// TIA Portal V16 program export: 5 tag tables, 70 data types, 8 data blocks, 77 code blocks (in call order from the OBs), 35 instance data blocks

VAR_GLOBAL   // PLC tag table "Default tag table"
   Tag_1 AT %M66.0 : Bool;
   Tag_2 AT %M60.0 : Bool;
   Tag_3 AT %M60.1 : Bool;
   Tag_4 AT %M60.2 : Bool;
   Tag_5 AT %M60.3 : Bool;
   Tag_6 AT %M70.0 : Bool;
   Tag_7 AT %M1.0 : Bool;
   Tag_8 AT %M1.1 : Bool;
   Tag_9 AT %M1.2 : Bool;
   Tag_10 AT %M70.1 : Bool;
   Tag_11 AT %M60.5 : Bool;
   Tag_12 AT %IW0 : Word;
   Tag_13 AT %IW2 : Word;
   Tag_14 AT %IW4 : Word;
   Tag_15 AT %M66.3 : Bool;
   Tag_16 AT %M17.0 : Bool;
   Tag_17 AT %M1717.0 : Bool;
   adım1 AT %M0.0 : Bool;
   step1 AT %M0.1 : Bool;
   step2 AT %M0.2 : Bool;
   step3 AT %M0.3 : Bool;
   step4 AT %M0.4 : Bool;
   step5 AT %M0.5 : Bool;
   Tag_18 AT %M170.0 : Bool;
   Tag_19 AT %M170.1 : Bool;
   step6 AT %M0.6 : Bool;
   step7 AT %M0.7 : Bool;
   Tag_20 AT %M1717.2 : Bool;
   Tag_21 AT %MD100 : DWord;
END_VAR

VAR_GLOBAL   // PLC tag table "LSimaHydTO_Constants"
END_VAR
VAR_GLOBAL CONSTANT   // user constants
   LSIMAHYD_PROFILE_POINTS_UPPER_LIMIT : Int := 20;   // Upper limit of the points in the force profile
   LSIMAHYD_VCHAR_POINTS_UPPER_LIMIT : Int := 40;   // Upper limit of the points in the valve characteristic
END_VAR

VAR_GLOBAL   // PLC tag table "SimaHydTO_HydAxisAnalog2_Interface"
   HydAxisAnalog_2_Sensor1_Interface_AddressIn AT %I1400.0 : "PD_TEL83_IN";   //    {ExternalWritable false}
   HydAxisAnalog_2_ForceSensor AT %IW1052 : Int;   //    {ExternalWritable false}
   HydAxisAnalog_2_Sensor1_Interface_AddressOut AT %Q1400.0 : "PD_TEL83_OUT";   //    {ExternalWritable false}
   HydAxisAnalog_2_OutputValue AT %QW2 : Int;   //    {ExternalWritable false}
END_VAR

VAR_GLOBAL   // PLC tag table "SimaHydTO_HydAxisAnalog_Interface"
   HydAxisAnalog_Sensor1_Interface_AddressIn AT %I1200.0 : "PD_TEL83_IN";   //    {ExternalWritable false}
   HydAxisAnalog_ForceSensor AT %IW1050 : Int;   //    {ExternalWritable false}
   HydAxisAnalog_Sensor1_Interface_AddressOut AT %Q1200.0 : "PD_TEL83_OUT";   //    {ExternalWritable false}
   HydAxisAnalog_OutputValue AT %QW0 : Int;   //    {ExternalWritable false}
END_VAR

VAR_GLOBAL   // PLC tag table "SimaHydTO_HydAxisServo_Interface"
   HydAxisServo_Actor_Interface_AddressIn AT %I1100.0 : "PD_TEL2_IN";   //    {ExternalWritable false}
   HydAxisServo_Sensor1_Interface_AddressIn AT %I1150.0 : "PD_TEL81_IN";   //    {ExternalWritable false}
   HydAxisServo_ForceSensor AT %IW1020 : Int;   //    {ExternalWritable false}
   HydAxisServo_Actor_Interface_AddressOut AT %Q1100.0 : "PD_TEL2_OUT";   //    {ExternalWritable false}
   HydAxisServo_Sensor1_Interface_AddressOut AT %Q1150.0 : "PD_TEL81_OUT";   //    {ExternalWritable false}
END_VAR

TYPE "LSimaHydTO_typeActor"
TITLE = LSimaHydTO_typeActor
// Actor configuration
// stored: IsFailsafeCompliant false
   STRUCT
      InverseDirection { S7_SetPoint := 'True'} : Bool := FALSE;   // Inversion of the setpoint if TRUE
      BiDirectional { S7_SetPoint := 'True'} : Bool := TRUE;   // Positive and negative outputs
      SubstituteValue { S7_SetPoint := 'True'} : LReal := 0.0;   // Substitute Output Value if disabled
      MaxDerivative { S7_SetPoint := 'True'} : LReal := 10000.0;   // Limit of changes at the manipulated variable
      DirectionValves { S7_SetPoint := 'True'} : "LSimaHydTO_typeActorDirectionValves";
   END_STRUCT;
END_TYPE

TYPE "LSimaHydTO_typeActorDirectionValves"
TITLE = LSimaHydTO_typeActorDirectionValves
// Settings of the direction valves control
// stored: IsFailsafeCompliant false
   STRUCT
      WaitTimeByDirectionChange { S7_SetPoint := 'True'} : LReal := 0.0;   // Waiting time between switching the digital valve valveForward and valveBackward for a direction change [s]
      DelayTimeValveForward { S7_SetPoint := 'True'} : LReal := 0.0;   // Reaction time for digital valve [s]
      DelayTimeValveBackward { S7_SetPoint := 'True'} : LReal := 0.0;   // Reaction time for digital valve [s]
      ValvesOffMode { S7_SetPoint := 'True'} : DInt := 0;   // 0: keep digital valves on after ramp down / 1: switch off digital valves after ramp down
      DisplacementForce { S7_SetPoint := 'True'} : Bool := FALSE;   // 1: force control by displacement ( inverse direction), e.g. die cushion
   END_STRUCT;
END_TYPE

TYPE "LSimaHydTO_typeAxisData"
TITLE = LSimaHydTO_typeAxisData
// Axis data
// stored: IsFailsafeCompliant false
   STRUCT
      Velocity : LReal := 0.0;   // Velocity setpoint
      Acceleration : LReal := 0.0;   // Setpoint acceleration
      Position : LReal := 0.0;   // Position setpoint
      Force : LReal := 0.0;   // Force setpoint
      ActualVelocity : LReal := 0.0;   // Actual velocity
      ActualSpeed : LReal := 0.0;   // Actual speed of the motor (only with PROFIdrive drive type)
      ActualAcceleration : LReal := 0.0;   // Actual acceleration
      ActualPosition : LReal := 0.0;   // Actual position
      ActualForce : LReal := 0.0;   // Actual force
      Actor { S7_SetPoint := 'True'} : "LSimaHydTO_typeActor";   // Actor configuration
      ValveCharacteristic { S7_SetPoint := 'True'} : "LSimaHydTO_typeValveCharacteristic";   // Valve characteristic
      ForceLimits { S7_SetPoint := 'True'} : "LSimaHydTO_typeForceLimits";   // Force limits
      Pressure_A_Transducer { S7_SetPoint := 'True'} : "LSimaHydTO_typeTransducer";   // Piston side pressure transducer configuration
      Pressure_B_Transducer { S7_SetPoint := 'True'} : "LSimaHydTO_typeTransducer";   // Piston rod side pressure transducer configuration
      PositionControl { S7_SetPoint := 'True'} : "LSimaHydTO_typePositionControl";   // Position control configuration data
      ForceControl { S7_SetPoint := 'True'} : "LSimaHydTO_typeForceControl";   // Force control configuration data
      DynamicAxisModel { S7_SetPoint := 'True'} : "LSimaHydTO_typeDynamicAxisModel";   // Settings of the balancing filter
      SmoothingFilter { S7_SetPoint := 'True'} : "LSimaHydTO_typeSmoothingFilter";   // Settings of the smoothing filter
      StatusActor { S7_SetPoint := 'True'} : "LSimaHydTO_typeStatusActor";   // Indicates the status of actor data
      StatusVChar { S7_SetPoint := 'True'} : "LSimaHydTO_typeStatusVChar";   // Indicates the status of valve characteristic data
      Status_A_Transducer { S7_SetPoint := 'True'} : "LSimaHydTO_typeStatusTransducer";   // Indicates the status of piston side pressure transducer data
      Status_B_Transducer { S7_SetPoint := 'True'} : "LSimaHydTO_typeStatusTransducer";   // Indicates the status of piston rod side pressure transducer data
      StatusServo { S7_SetPoint := 'True'} : "LSimaHydTO_typeStatusServo";   // Indicates the status of position control
      StatusForce { S7_SetPoint := 'True'} : "LSimaHydTO_typeStatusForce";   // Indicates the status of force control
      StatusForceProfile { S7_SetPoint := 'True'} : "LSimaHydTO_typeStatusForceProfile";   // Indicates the status of a force profile processing
      ErrorWord : DWord;   // Error information
      ErrorDetail { S7_SetPoint := 'True'} : "LSimaHydTO_typeErrorDetail";   // Error Details
      "Name" { S7_SetPoint := 'True'} : WString[24];   // Name displayed on HMI
      TO_Axis : DB_ANY;   // Number of connected technology object (TO)
      DataInitialized : Bool;   // Axis data completely initialized
      Internal { S7_SetPoint := 'True'} : "LSimaHydTO_typeInternal";   // Internal axis data
   END_STRUCT;
END_TYPE

TYPE "LSimaHydTO_typeDynamicAxisModel"
TITLE = LSimaHydTO_typeDynamicAxisModel
// Settings of the balancing filter
// stored: IsFailsafeCompliant false
   STRUCT
      VelocityTimeConstant { S7_SetPoint := 'True'} : LReal;   // Speed control loop substitute time [s]
      ForceTimeConstant { S7_SetPoint := 'True'} : LReal;   // Force control loop substitute time [s]
   END_STRUCT;
END_TYPE

TYPE "LSimaHydTO_typeDynamicLimits"
TITLE = LSimaHydTO_typeDynamicLimits
// Dynamic limits
// stored: IsFailsafeCompliant false
   STRUCT
      MaxVelocity { S7_SetPoint := 'True'} : LReal := 500.0;   // Maximum permissible velocity of the axis
      MaxAcceleration { S7_SetPoint := 'True'} : LReal := 10000.0;   // Maximum permissible acceleration of the axis
      MaxDeceleration { S7_SetPoint := 'True'} : LReal := 10000.0;   // Maximum permissible deceleration of the axis
      MaxJerk { S7_SetPoint := 'True'} : LReal := 200000.0;   // Maximum permissible jerk on the axis/ not used yet
   END_STRUCT;
END_TYPE

TYPE "LSimaHydTO_typeErrorDetail"
TITLE = LSimaHydTO_typeErrorDetail
// Error Details
// stored: IsFailsafeCompliant false
   STRUCT
      Number : UDInt;   // Alarm number
      Reaction : DInt;   // Effective alarm reaction
   END_STRUCT;
END_TYPE

TYPE "LSimaHydTO_typeForceControl"
TITLE = LSimaHydTO_typeForceControl
// Force control configuration data
// stored: IsFailsafeCompliant false
   STRUCT
      SmoothingTimeByChangeDifference { S7_SetPoint := 'True'} : LReal;   // Time constant for smoothing manipulated variable jumps
      PreControl { S7_SetPoint := 'True'} : LReal := 0.0;   // Weighting factor of the precontrol Kpc [%]
      Stiffness { S7_SetPoint := 'True'} : LReal;   // Stiffness of the system, should be > 0.0 if preControl is used
      ProportionalGain { S7_SetPoint := 'True'} : LReal := 1.0;   // Proportional gain Kp
      IntegralTime { S7_SetPoint := 'True'} : LReal;   // Active integral action time Ti [s]
      DerivativeTime { S7_SetPoint := 'True'} : LReal;   // Active derivative action time Td [s]
      DecayTime { S7_SetPoint := 'True'} : LReal := 0.0;   // Decay time constant of the DT1 component [s]
      OutputUppLimit { S7_SetPoint := 'True'} : LReal := 10000.0;   // Manipulated value high limit
      OutputLowLimit { S7_SetPoint := 'True'} : LReal := -10000.0;   // Manipulated value low limit
      SmoothSwitching { S7_SetPoint := 'True'} : Bool := TRUE;   // Switching mode to force control, if TRUE, initial command value of the force controller will be presetted for edgeless valve setpoint
      InvertSetpoint { S7_SetPoint := 'True'} : Bool;   // Invert output of controller if TRUE
   END_STRUCT;
END_TYPE

TYPE "LSimaHydTO_typeForceLimits"
TITLE = LSimaHydTO_typeForceLimits
// Force limits
// stored: IsFailsafeCompliant false
   STRUCT
      MaxForce { S7_SetPoint := 'True'} : LReal := 100.0;   // Maximum force
      MaxForceRamp { S7_SetPoint := 'True'} : LReal := 10000.0;   // Force increase limitation
   END_STRUCT;
END_TYPE

TYPE "LSimaHydTO_typeInternal"
TITLE = LSimaHydTO_typeInternal
// Internal axis data
// stored: IsFailsafeCompliant false
   STRUCT
      Control { S7_SetPoint := 'True'} : "LSimaHydTO_typeInternalControl";   // Command structure, use for axis control
      MotionData { S7_SetPoint := 'True'} : "LSimaHydTO_typeInternalMotionData";   // Motion command data
      PositionLimits_SW { S7_SetPoint := 'True'} : "LSimaHydTO_typePositionLimits";   // Software position limit switch
      UnitsCorrection { S7_SetPoint := 'True'} : "LSimaHydTO_typeInternalUnitsCorrection";   // Correction of units
      CommandIDPool { ExternalAccessible := 'False'; ExternalVisible := 'False'; ExternalWritable := 'False'} : UDInt;   // Source for unique command ID's
   END_STRUCT;
END_TYPE

TYPE "LSimaHydTO_typeInternalCmdTracking"
TITLE = LSimaHydTO_typeInternalCmdTracking
// Command tracking
// stored: IsFailsafeCompliant false
   STRUCT
      CommandID : UDInt := 0;   // Command ID for tracking
      State : Word := 0;   // Command state
   END_STRUCT;
END_TYPE

TYPE "LSimaHydTO_typeInternalControl"
TITLE = LSimaHydTO_typeInternalControl
// Command structure, use for axis control
// stored: IsFailsafeCompliant false
   STRUCT
      AckError : Bool;   // Acknowledge error of axis
      ExecuteForceLimiting : Bool;   // Rising edge starts force limiting defined by ForceCommand
      ExecuteForceControl : Bool;   // Rising edge starts force control defined by ForceCommand
      RequestForward : Bool;   // request to open direction valve forward
      RequestBackward : Bool;   // request to open direction valve backward
      ForceCommand { S7_SetPoint := 'True'} : "LSimaHydTO_typeInternalControlForceCmd";   // Defines force command
      DirectOutput { S7_SetPoint := 'True'} : "LSimaHydTO_typeInternalControlDirectOutput";
   END_STRUCT;
END_TYPE

TYPE "LSimaHydTO_typeInternalControlDirectOutput"
TITLE = LSimaHydTO_typeInternalControlDirectOutput
// Manual output control
// stored: IsFailsafeCompliant false
   STRUCT
      activate : Bool;   // enables direct setting of output
      jogForward : Bool;   // direct output is active in positive direction if TRUE
      jogBackward : Bool;   // direct output is active in negative direction if TRUE
      commandValueForward : LReal := 5.0;   // direct output value in positive direction [%]
      commandValueBackward : LReal := 5.0;   // direct output value in negative direction [%]
      commandValueRamp : LReal := 100.0;   // Ramp for command value [%/s]
      offset : LReal := 0.0;   // Manipulated variable as drift compensation [%]
      safetyDistance : LReal := 50.0;   // Safety distance to avoid passing over the min. and max. positions [mm]
      commandID : UDInt;   // commanID for tracking
   END_STRUCT;
END_TYPE

TYPE "LSimaHydTO_typeInternalControlForceCmd"
TITLE = LSimaHydTO_typeInternalControlForceCmd
// Defines force command
// stored: IsFailsafeCompliant false
   STRUCT
      mode : DInt;   // 0: deactivate / 1: activate immediately / 2: starting from the time a condition is met.
      forceProfileMode : DInt;   // 0: with force value / 1: profile is a function of time / 2: profile is a function of position
      conditionMode : DInt := 1;   // 1: based on time / 2: based on position / 3: based on force/pressure
      compareMode : DInt := 1;   // 1: Value greater than or equal to ConditionValue / 2: Value less than ConditionValue
      conditionValue : LReal;   // comparison value for switching condition
      clampingMonitoring : Bool;   // TRUE: end stop detection is activated, motion stops after detection
      followingErrorDeviation : LReal;   // Required following error for recognition of the endstop
      forceValue : LReal;   // Force setpoint
      forceRamp : LReal;   // Force setpoint increase
      velocityLimitingValue : LReal;   // Rate limiting value during pressure control, the dynamic response of the pressure Value > 0.0 Use the specified value
      commandID : UDInt;   // commanID for tracking
   END_STRUCT;
END_TYPE

TYPE "LSimaHydTO_typeInternalMotionData"
TITLE = LSimaHydTO_typeInternalMotionData
// Motion command data
// stored: IsFailsafeCompliant false
   STRUCT
      PositionControlled : Bool := FALSE;   // Activates position controller
      ForceLimited : Bool := FALSE;   // Enable force limiting
      ForceControlled : Bool := FALSE;   // Enable force control
      RampingForward : Bool;   // enable signal for ramping in positive direction
      RampingBackward : Bool;   // enable signal for ramping in negative direction
      ForceCmdTracking { S7_SetPoint := 'True'} : "LSimaHydTO_typeInternalCmdTracking";   // Force command tracking
      DirectOutput { S7_SetPoint := 'True'} : "LSimaHydTO_typeInternalStatusDirectOutput";
   END_STRUCT;
END_TYPE

TYPE "LSimaHydTO_typeInternalStatusDirectOutput"
TITLE = LSimaHydTO_typeInternalStatusDirectOutput
// Manual output control
// stored: IsFailsafeCompliant false
   STRUCT
      active : Bool;   // displays activity of manual output operation
      rampingDown : Bool;   // ramping down due to positioning limits
      minSafetyPositionOverrun : Bool;   // the min. safety position was passed
      maxSafetyPositionOverrun : Bool;   // the max. safety position was passed
      QOutputValue : LReal;
      cmdTracking { S7_SetPoint := 'True'} : "LSimaHydTO_typeInternalCmdTracking";
   END_STRUCT;
END_TYPE

TYPE "LSimaHydTO_typeInternalUnitsCorrection"
TITLE = LSimaHydTO_typeInternalUnitsCorrection
// stored: IsFailsafeCompliant false
   STRUCT
      velFactor : LReal := 1.0;
      accFactor : LReal := 1.0;
   END_STRUCT;
END_TYPE

TYPE "LSimaHydTO_typeMeasuredValues"
TITLE = LSimaHydTO_typeMeasuredValues
// Measurement results
// stored: IsFailsafeCompliant false
   STRUCT
      forward { S7_SetPoint := 'True'} : "LSimaHydTO_typeVCharMeasured";   // measured values in positive direction
      backward { S7_SetPoint := 'True'} : "LSimaHydTO_typeVCharMeasured";   // measured values in negative direction
   END_STRUCT;
END_TYPE

TYPE "LSimaHydTO_typeMeasurementConfig"
TITLE = LSimaHydTO_typeMeasurementConfig
// Configuration of the measurement function
// stored: IsFailsafeCompliant false
   STRUCT
      waitTimeMeasurement { S7_SetPoint := 'True'} : DInt := 100;   // Waiting time after ramping [ms]
      maxMeasurementTime { S7_SetPoint := 'True'} : DInt := 200;   // Measurement time [ms]
      offset { S7_SetPoint := 'True'} : LReal;   // Manipulated variable as drift compensation [%]
      safetyDistance { S7_SetPoint := 'True'} : LReal;   // Safety distance to avoid passing over the min. and max. positions
      forward { S7_SetPoint := 'True'} : "LSimaHydTO_typeMeasurementQOutput";   // Structure to define the manipulated variable
      backward { S7_SetPoint := 'True'} : "LSimaHydTO_typeMeasurementQOutput";   // Structure to define the manipulated variable
      numberOfRetryMeasurement { S7_SetPoint := 'True'} : Int := 1;   // Number of repeat attempts to measure the velocity, this parameter should be greater than / equal to 1
   END_STRUCT;
END_TYPE

TYPE "LSimaHydTO_typeMeasurementQOutput"
TITLE = LSimaHydTO_typeMeasurementQOutput
// Structure to define the manipulated variable
// stored: IsFailsafeCompliant false
   STRUCT
      enableMeasurement { S7_SetPoint := 'True'} : Bool := TRUE;   // Enables measurement in this direction
      maxVelocity { S7_SetPoint := 'True'} : Real := 500.0;   // Velocity limit in this direction
      setpointForMovement { S7_SetPoint := 'True'} : Real := 40.0;   // Substitute value for movements if a measurement is not active [%]
      ramp { S7_SetPoint := 'True'} : Real := 100.0;   // manipulated variable – increase/decrease [%/s]
      minQOutputValue { S7_SetPoint := 'True'} : Real;   // start measurement with this value
      fineRange { S7_SetPoint := 'True'} : "LSimaHydTO_typeMeasurementQOutputRange";   // measurement in the fine area
      coarseRange { S7_SetPoint := 'True'} : "LSimaHydTO_typeMeasurementQOutputRange";   // measurement in the coarse area
   END_STRUCT;
   // fineRange.maxQOutputValue := 40.0;
   // fineRange.numberOfPoints := 10;
   // coarseRange.maxQOutputValue := 100.0;
   // coarseRange.numberOfPoints := 10;
END_TYPE

TYPE "LSimaHydTO_typeMeasurementQOutputRange"
TITLE = LSimaHydTO_typeMeasurementQOutputRange
// stored: IsFailsafeCompliant false
   STRUCT
      maxQOutputValue { S7_SetPoint := 'True'} : Real;   // incremented up to this value
      numberOfPoints { S7_SetPoint := 'True'} : Int;   // number of points for this range
   END_STRUCT;
END_TYPE

TYPE "LSimaHydTO_typeMotionVector"
TITLE = LSimaHydTO_typeMotionVector
// Values of a motion vector
// stored: IsFailsafeCompliant false
   STRUCT
      Position : LReal;   // Position
      Velocity : LReal;   // Velocity
      Acceleration : LReal;   // Acceleration
   END_STRUCT;
END_TYPE

TYPE "LSimaHydTO_typePositionControl"
TITLE = LSimaHydTO_typePositionControl
// Position control configuration data
// stored: IsFailsafeCompliant false
   STRUCT
      SmoothingTimeByChangeDifference { S7_SetPoint := 'True'} : LReal;   // Time constant for smoothing manipulated variable jumps [s]
      PreControl { S7_SetPoint := 'True'} : LReal := 100.0;   // Weighting factor of the precontrol Kpc [%]
      ProportionalGain { S7_SetPoint := 'True'} : LReal := 10.0;   // Proportional gain Kp [1/s]
      IntegralTime { S7_SetPoint := 'True'} : LReal;   // Active integral action time Ti [s]
      DerivativeTime { S7_SetPoint := 'True'} : LReal;   // Active derivative action time Td [s]
      DecayTime { S7_SetPoint := 'True'} : LReal := 0.0;   // Decay time constant of the DT1 component [s]
      OutputUppLimit { S7_SetPoint := 'True'} : LReal := 10000.0;   // Manipulated value high limit [unit/s]
      OutputLowLimit { S7_SetPoint := 'True'} : LReal := -10000.0;   // Manipulated value low limit [unit/s]
   END_STRUCT;
END_TYPE

TYPE "LSimaHydTO_typePositionLimits"
TITLE = LSimaHydTO_typePositionLimits
// Software position limit switch
// stored: IsFailsafeCompliant false
   STRUCT
      Active { S7_SetPoint := 'True'} : Bool := TRUE;   // FALSE: Monitoring disabled / TRUE: Monitoring enabled
      MinPosition { S7_SetPoint := 'True'} : LReal := -1000000000000.0;   // Position of negative SW limit switch
      MaxPosition { S7_SetPoint := 'True'} : LReal := 1000000000000.0;   // Position of positive SW limit switch
   END_STRUCT;
END_TYPE

TYPE "LSimaHydTO_typeProfile"
TITLE = LSimaHydTO_typeProfile
// Configuration for the profile point
// stored: IsFailsafeCompliant false
   STRUCT
      LeadingValue { S7_SetPoint := 'True'} : Array[0.."LSIMAHYD_PROFILE_POINTS_UPPER_LIMIT"] of Real;   // Input values array
      Value { S7_SetPoint := 'True'} : Array[0.."LSIMAHYD_PROFILE_POINTS_UPPER_LIMIT"] of Real;   // Output values array
      MaxIdx { S7_SetPoint := 'True'} : Int;   // Max used index in arrays
   END_STRUCT;
END_TYPE

TYPE "LSimaHydTO_typeSmoothingFilter"
TITLE = LSimaHydTO_typeSmoothingFilter
// Settings of the smoothing filter
// stored: IsFailsafeCompliant false
   STRUCT
      VelocityFilter { S7_SetPoint := 'True'} : LReal := 0.0;   // Time constant for actual velocity smoothing filter [s]
      AccelerationFilter { S7_SetPoint := 'True'} : LReal := 0.0;   // Time constant for actual acceleration smoothing filter [s]
   END_STRUCT;
END_TYPE

TYPE "LSimaHydTO_typeStatusActor"
TITLE = LSimaHydTO_typeStatusActor
// Indicates the status of actor data
// stored: IsFailsafeCompliant false
   STRUCT
      SetPoint : LReal := 0.0;   // Manipulated variable
      AddSetPoint : LReal := 0.0;   // Additional setpoint
      QOutputValue : LReal := 0.0;   // Output value in relation to Q-output [%]
      Enabled : Bool;   // Output is enabled
      ValveForward : Bool := FALSE;   // Control bit for positive direction
      ValveBackward : Bool := FALSE;   // Control bit for negative direction
   END_STRUCT;
END_TYPE

TYPE "LSimaHydTO_typeStatusForce"
TITLE = LSimaHydTO_typeStatusForce
// Indicates the status of force control
// stored: IsFailsafeCompliant false
   STRUCT
      ForceLimitingCommand { ExternalWritable := 'False'} : Bool;   // TRUE: Axis is in force limiting mode; FALSE: Axis isn't in force limiting mode/ SimaHyd only
      InLimitation { ExternalWritable := 'False'} : Bool;   // TRUE: Axis is operating at the force limit; FALSE: axis is not operating at the force limit/ SimaHyd only
      InClamping { ExternalWritable := 'False'} : Bool;   // TRUE: Axis is clamped at a fixed stop; FALSE: Axis is not clamped at a fixed stop
      ForceControl { ExternalWritable := 'False'} : Bool;   // TRUE: Axis is in force control mode; FALSE: Axis isn't in force control mode/ SimaHyd only
      TargetForce { ExternalWritable := 'False'} : LReal;   // Target force
      ForceDerivedValue { ExternalWritable := 'False'} : LReal;   // Rate-of-change limiting for the force setpoint
      PreControlValue { ExternalWritable := 'False'} : LReal;   // Force precontrol value
      BalancedForce { ExternalWritable := 'False'} : LReal;   // Force after the balancing filter
      ControlDifference { ExternalWritable := 'False'} : LReal;   // Control error
      ControlOutput { ExternalWritable := 'False'} : LReal;   // Control variable
   END_STRUCT;
END_TYPE

TYPE "LSimaHydTO_typeStatusForceProfile"
TITLE = LSimaHydTO_typeStatusForceProfile
// Indicates the status of a force profile processing
// stored: IsFailsafeCompliant false
   STRUCT
      ActualProfile : UInt := 0;   // Currently effective force profile DB number
      ForceProfileMode : DInt := 0;   // 0: with force value / 1: profile is a function of time / 2: profile is a function of position
      Active : Bool := FALSE;   // Activation status of a command for specifying the force profile
      State : DInt := 0;   // Execution state: 0: inactive / 1: in interpolation / 2: on profile / 3: profile end
      BaseValue : LReal := 0.0;   // Current reference value
      ProfileValue : LReal := 0.0;   // Profile value for the base value
   END_STRUCT;
END_TYPE

TYPE "LSimaHydTO_typeStatusServo"
TITLE = LSimaHydTO_typeStatusServo
// Indicates the status of position control
// stored: IsFailsafeCompliant false
   STRUCT
      BalancedPosition { ExternalWritable := 'False'} : LReal;   // Position after the balancing filter
      ControlDifference { ExternalWritable := 'False'} : LReal;   // Control error
   END_STRUCT;
END_TYPE

TYPE "LSimaHydTO_typeStatusTransducer"
TITLE = LSimaHydTO_typeStatusTransducer
// Indicates the status of transducer data
// stored: IsFailsafeCompliant false
   STRUCT
      RawValue : Word;   // Raw data of analog input
      PressureValue : LReal;   // actual pressure In pressure units
      ForceValue : LReal;   // actual force In force units
      Error : Bool := FALSE;   // Indicates error of transducer
   END_STRUCT;
END_TYPE

TYPE "LSimaHydTO_typeStatusVChar"
TITLE = LSimaHydTO_typeStatusVChar
// Indicates the status of valve characteristic data
// stored: IsFailsafeCompliant false
   STRUCT
      ActualVChar : UInt := 0;   // Currently effective valve characteristic DB number
   END_STRUCT;
END_TYPE

TYPE "LSimaHydTO_typeTransducer"
TITLE = LSimaHydTO_typeTransducer
// Pressure transducer configuration
// stored: IsFailsafeCompliant false
   STRUCT
      HWReference { S7_SetPoint := 'True'} : Int := 16#6C00;   // Normalization of the raw value for 100%. Distinction between a SIMATIC or a SINAMICS periphery: SIMATIC = 27648, SINAMICS = 16384
      NominalPressure { S7_SetPoint := 'True'} : LReal := 400.0;   // Nominal pressure of transducer, e.g. 400 [bar]
      Area { S7_SetPoint := 'True'} : LReal := 1.0;   // Area [mm2] or [in2]
      Offset { S7_SetPoint := 'True'} : LReal := 0.0;   // Offset in pressure units
      FilterTime { S7_SetPoint := 'True'} : LReal := 0.0;   // Smoothing filter
      ErrorValue { S7_SetPoint := 'True'} : Word := 16#7FFF;   // Error signal
   END_STRUCT;
END_TYPE

TYPE "LSimaHydTO_typeVCharData"
TITLE = LSimaHydTO_typeVCharData
// Valve characteristic description
// stored: IsFailsafeCompliant false
   STRUCT
      QOutput { S7_SetPoint := 'True'} : Array[0.."LSIMAHYD_VCHAR_POINTS_UPPER_LIMIT"] of Real;   // Output values array
      Velocity { S7_SetPoint := 'True'} : Array[0.."LSIMAHYD_VCHAR_POINTS_UPPER_LIMIT"] of Real;   // Velocity values array
      VelocityLimitPositive { S7_SetPoint := 'True'} : Real;   // Max velocity in positive direction
      VelocityLimitNegative { S7_SetPoint := 'True'} : Real;   // Max velocity in negative direction
      ZeroZonePositive { S7_SetPoint := 'True'} : Real;   // Overlapping zone of valve in positive direction
      ZeroZoneNegative { S7_SetPoint := 'True'} : Real;   // Overlapping zone of valve in negative direction
      MaxIdx { S7_SetPoint := 'True'} : Int;   // Max used index in arrays
      "Name" { S7_SetPoint := 'True'} : WString[24];   // Symbolic name displayed on HMI for index of array
   END_STRUCT;
END_TYPE

TYPE "LSimaHydTO_typeVCharMeasured"
TITLE = LSimaHydTO_typeVCharMeasured
// Measured Values in one direction
// stored: IsFailsafeCompliant false
   STRUCT
      qOutput : Array[0.."LSIMAHYD_VCHAR_POINTS_UPPER_LIMIT"] of Real;   // manipulated variable
      velocity : Array[0.."LSIMAHYD_VCHAR_POINTS_UPPER_LIMIT"] of Real;   // velocity
      maxVelocity : Real;   // max. measured velocity
      minQOutput : Real;   // min. manipulated variable
      maxQOutput : Real;   // max. manipulated variable
      maxIndexMeasurement : Int;   // measurement was made up to this index
      coarseBegin : Real;   // coarse area begins by this index
   END_STRUCT;
END_TYPE

TYPE "LSimaHydTO_typeValveCharacteristic"
TITLE = LSimaHydTO_typeValveCharacteristic
// Valve characteristic
// stored: IsFailsafeCompliant false
   STRUCT
      DB_NUMBER { S7_SetPoint := 'True'} : UInt;   // Number of DB of type LSimaHydTO_typeVCharData with valve profile data
      SmoothChangeTime { S7_SetPoint := 'True'} : Real;   // Filter time for smooth changing
      SmoothingMode { S7_SetPoint := 'True'} : Int;   // Filter mode for smooth changing: 0: T1 / 1: ramping with constant ramp / 2: ramping with time
   END_STRUCT;
END_TYPE

TYPE "SimaHydTO_typeAxesArray"
TITLE = SimaHydTO_typeAxesArray
// Axis array of HMI axis selection
// stored: IsFailsafeCompliant false
   STRUCT
      axisData { ExternalAccessible := 'False'; ExternalVisible := 'False'; ExternalWritable := 'False'} : DB_ANY;   // DB number of hydraulic axis DB (HydAxisTO)
      basicControl { ExternalAccessible := 'False'; ExternalVisible := 'False'; ExternalWritable := 'False'; S7_SetPoint := 'True'} : "SimaHydTO_typeHMIConnectionBasicAxisControlCommand";   // HMI -> PLC: Axis commands of technology object via PLCopen functions
      directOutputControl { ExternalAccessible := 'False'; ExternalVisible := 'False'; ExternalWritable := 'False'; S7_SetPoint := 'True'} : "SimaHydTO_typeIHMIConnectionBasicAxisControlDirectOutput";
      VCharMeasurement { ExternalAccessible := 'False'; ExternalVisible := 'False'; ExternalWritable := 'False'; S7_SetPoint := 'True'} : "SimaHydTO_typeAxesArrayVCharMeasurement";
      advancedControl { ExternalAccessible := 'False'; ExternalVisible := 'False'; ExternalWritable := 'False'; S7_SetPoint := 'True'} : "SimaHydTO_typeHMIConnectionAdvancedAxisControlCommand";   // Advanced axis commands of technology object via PLCopen functions
      initialized { ExternalAccessible := 'False'; ExternalVisible := 'False'; ExternalWritable := 'False'} : Bool;   // Axis data initialized
   END_STRUCT;
END_TYPE

TYPE "SimaHydTO_typeAxesArrayVCharMeasurement"
TITLE = SimaHydTO_typeAxesArrayVCharMeasurement
// Axis array of HMI axis selection
// stored: IsFailsafeCompliant false
   STRUCT
      requestForward { ExternalAccessible := 'False'; ExternalVisible := 'False'; ExternalWritable := 'False'} : Bool;   // Switches the digital valves to move in the positive direction
      requestBackward { ExternalAccessible := 'False'; ExternalVisible := 'False'; ExternalWritable := 'False'} : Bool;   // Switches the digital valves to move in the negative direction
      enableRampingForward { ExternalAccessible := 'False'; ExternalVisible := 'False'; ExternalWritable := 'False'} : Bool := True;   // Enable ramping of Q-Output value (voltage) in positivedirection
      enableRampingBackward { ExternalAccessible := 'False'; ExternalVisible := 'False'; ExternalWritable := 'False'} : Bool := True;   // Enable ramping of Q-Output value (voltage) in negative direction
   END_STRUCT;
END_TYPE

TYPE "SimaHydTO_typeHMIConnection"
TITLE = SimaHydTO_typeHMIConnection
// HMI connection interface data block
// stored: IsFailsafeCompliant false
   STRUCT
      AxisData { S7_SetPoint := 'True'} : "SimaHydTO_typeHMIConnectionAxisData";
      AxisToData { S7_SetPoint := 'True'} : "SimaHydTO_typeHMIConnectionAxisToData";
      AxisSelector { S7_SetPoint := 'True'} : "SimaHydTO_typeHMIConnectionAxisSelector";
      BasicAxisControl { S7_SetPoint := 'True'} : "SimaHydTO_typeHMIConnectionBasicAxisControl";
      GetCharacteristics { S7_SetPoint := 'True'} : "SimaHydTO_typeHMIConnectionGetCharacteristicInterface";
      HmiData { S7_SetPoint := 'True'} : "SimaHydTO_typeHMIConnectionHmiData";
      VCharEditor { S7_SetPoint := 'True'} : "SimaHydTO_typeHMIConnectionVCharEditor";
      AdvancedAxisControl { S7_SetPoint := 'True'} : "SimaHydTO_typeHMIConnectionAdvancedAxisControl";
      ParameterSettings { S7_SetPoint := 'True'} : "SimaHydTO_typeHMIConnectionParameterSettings";
   END_STRUCT;
END_TYPE

TYPE "SimaHydTO_typeHMIConnectionAdvancedAxisControl"
TITLE = SimaHydTO_typeHMIConnectionAdvancedAxisControl
// HMI interface: Advanced axis control
// stored: IsFailsafeCompliant false
   STRUCT
      Command { S7_SetPoint := 'True'} : "SimaHydTO_typeHMIConnectionAdvancedAxisControlCommand";   // Command (HMI -> PLC)
      Status { S7_SetPoint := 'True'} : "SimaHydTO_typeHMIConnectionAdvancedAxisControlStatus";   // Status (PLC -> HMI)
   END_STRUCT;
END_TYPE

TYPE "SimaHydTO_typeHMIConnectionAdvancedAxisControlCommand"
TITLE = SimaHydTO_typeHMIConnectionAdvancedAxisControlCommand
// HMI interface: Advanced axis control
// stored: IsFailsafeCompliant false
   STRUCT
      moveRelativeExecute : Bool;   // MC_MoveRelative: Start job with a positive edge
      moveRelativeDistance : LReal;   // Distance of relative movement
      moveAbsoluteExecute : Bool;   // MC_MoveAbsolute: Start job with a positive edge
      moveAbsolutePosition : LReal;   // Target position of absolute movement
      moveAbsoluteDirection : Int := 3;   // Direction of absolute movement: 0: Positive direction / 1: Negative direction / 3: Shortest direction
      haltExecute : Bool;   // MC_Halt: Start job with a positive edge
      haltAbortAcceleration : Bool;   // Acceleration control: False: The current acceleration at the start of the job is reduced using the configured jerk. Afterwards, the deceleration builds up / True: The acceleration is set to 0.0 at the start of the job, and the deceleration immediately builds up.
      Velocity : LReal := -1.0;   // Velocity of movement
      Acceleration : LReal := -1.0;   // Acceleration of movement
      Deceleration : LReal := -1.0;   // Deceleration of movement
      Jerk : LReal := -1.0;   // Jerk of movement
   END_STRUCT;
END_TYPE

TYPE "SimaHydTO_typeHMIConnectionAdvancedAxisControlStatus"
TITLE = SimaHydTO_typeHMIConnectionAdvancedAxisControlStatus
// HMI interface: Advanced axis control
// stored: IsFailsafeCompliant false
   STRUCT
      moveRelativeDone : Bool;   // MC_MoveRelative: Job is completed
      moveRelativeBusy : Bool;   // MC_MoveRelative: Job is running
      moveAbsoluteDone : Bool;   // MC_MoveAbsolute: Job is completed
      moveAbsoluteBusy : Bool;   // MC_MoveAbsolute: Job is running
      haltDone : Bool;   // MC_Halt: Job is running
      haltBusy : Bool;   // MC_Halt: Job is running
      commandAborted : Bool;   // The job was aborted by another job during execution (see also StatusID)
      error : Bool;   // An error occurred during execution of the job. The job is rejected. The cause of the error can be found in the "ErrorID" parameter.
      errorID : Word;   // ErrorID of motion control instruction (see also StatusID)
      statusID : Int;   // Additional specification of affected Motion control instruction of CommandAborted or Error: 0: No instruction / 1: MC_MoveRelative / 2: MC_MoveAbsolute / 3: MC_Halt
   END_STRUCT;
END_TYPE

TYPE "SimaHydTO_typeHMIConnectionAxisData"
TITLE = SimaHydTO_typeHMIConnectionAxisData
// Axis data
// stored: IsFailsafeCompliant false
   STRUCT
      Velocity : LReal := 0.0;   // Velocity setpoint
      Acceleration : LReal := 0.0;   // Setpoint acceleration
      Position : LReal := 0.0;   // Position setpoint
      Force : LReal := 0.0;   // Force setpoint
      ActualVelocity : LReal := 0.0;   // Actual velocity
      ActualSpeed : LReal := 0.0;   // Actual speed of the motor (only with PROFIdrive drive type)
      ActualAcceleration : LReal := 0.0;   // Actual acceleration
      ActualPosition : LReal := 0.0;   // Actual position
      ActualForce : LReal := 0.0;   // Actual force
      StatusActor { S7_SetPoint := 'True'} : "LSimaHydTO_typeStatusActor";   // Indicates the status of actor data
      StatusVChar { S7_SetPoint := 'True'} : "LSimaHydTO_typeStatusVChar";   // Indicates the status of valve characteristic data
      Status_A_Transducer { S7_SetPoint := 'True'} : "LSimaHydTO_typeStatusTransducer";   // Indicates the status of piston side pressure transducer data
      Status_B_Transducer { S7_SetPoint := 'True'} : "LSimaHydTO_typeStatusTransducer";   // Indicates the status of piston rod side pressure transducer data
      StatusServo { S7_SetPoint := 'True'} : "LSimaHydTO_typeStatusServo";   // Indicates the status of position control
      StatusForce { S7_SetPoint := 'True'} : "LSimaHydTO_typeStatusForce";   // Indicates the status of force control
      StatusForceProfile { S7_SetPoint := 'True'} : "LSimaHydTO_typeStatusForceProfile";   // Indicates the status of a force profile processing
      ErrorWord : DWord;   // Error information
      ErrorDetail { S7_SetPoint := 'True'} : "LSimaHydTO_typeErrorDetail";   // Error Details
      "Name" : WString[24];   // Name displayed on HMI
   END_STRUCT;
END_TYPE

TYPE "SimaHydTO_typeHMIConnectionAxisSelector"
TITLE = SimaHydTO_typeHMIConnectionAxisSelector
// HMI interface: Axis selection of axis array
// stored: IsFailsafeCompliant false
   STRUCT
      Command { S7_SetPoint := 'True'} : "SimaHydTO_typeHMIConnectionAxisSelectorCommand";   // Data: HMI -> PLC
      Status { S7_SetPoint := 'True'} : "SimaHydTO_typeHMIConnectionAxisSelectorStatus";   // Data: PLC -> HMI
   END_STRUCT;
END_TYPE

TYPE "SimaHydTO_typeHMIConnectionAxisSelectorCommand"
TITLE = SimaHydTO_typeHMIConnectionAxisSelectorCommand
// HMI interface: Axis selection of axis array - Command (HMI -> PLC)
// stored: IsFailsafeCompliant false
   STRUCT
      previousObject : Bool;
      nextObject : Bool;
      executeDirectIndexSelection : Bool;
      directIndexSelection : Int;
   END_STRUCT;
END_TYPE

TYPE "SimaHydTO_typeHMIConnectionAxisSelectorStatus"
TITLE = SimaHydTO_typeHMIConnectionAxisSelectorStatus
// HMI interface: Axis selection of axis array - Status (PLC -> HMI)
// stored: IsFailsafeCompliant false
   STRUCT
      actualAxisIndex : Int;   // Actual selected array index
      selectedAxis : DB_ANY;   // DB number of actual selected hydraulic axis
      selectedTO_Axis : DB_ANY;   // DB/TO number of actual selected technology object axis
      selectedVChar : DB_ANY;   // DB number of actual selected valve characteristics
      selectedAxisInteger : UInt;   // DB number of actual selected hydraulic axis as integer value
      selectedAxisTOInteger : UInt;   // DB/TO number of actual selected technology object as integer value
      selectedVCharInteger : UInt;   // DB number of actual selected valve characteristics as integer value
      selectedAxisName : WString[24];   // Name of actual selected hydraulic axis
      selectedVCharName : WString[24];   // Name of active VChat of selected hydraulic axis
      selectedTypeOfAxis : Int;   // 0: No axis / 1: Speed axis / 2: Positioning axis / 3: Synchronous axis / 4: External encoder
      selectionChanged : Bool;   // axis selection is changed
      dataValid : Bool;   // Selected data valid
      dataError : Bool;   // Error of data selection
   END_STRUCT;
END_TYPE

TYPE "SimaHydTO_typeHMIConnectionAxisToData"
TITLE = SimaHydTO_typeHMIConnectionAxisToData
// HMI interface: Technology object axis diagnostic words
// stored: IsFailsafeCompliant false
   STRUCT
      statusWord : DWord;
      warningWord : DWord;
      errorWord : DWord;
      errorDetail { S7_SetPoint := 'True'} : "SimaHydTO_typeHMIConnectionAxisToDataErrorDetail";
      axisUnits { S7_SetPoint := 'True'} : "SimaHydTO_typeHMIConnectionAxisToDataAxisUnits";
      typeOfAxis : Int;   // 0: No axis / 1: Speed axis / 2: Positioning axis / 3: Synchronous axis / 4: External encoder
   END_STRUCT;
END_TYPE

TYPE "SimaHydTO_typeHMIConnectionAxisToDataAxisUnits"
TITLE = SimaHydTO_typeHMIConnectionAxisToDataAxisUnits
// HMI interface: Technology object axis units
// stored: IsFailsafeCompliant false
   STRUCT
      lengthUnit : UDInt := 0;
      velocityUnit : UDInt := 0;
      forceUnit : UDInt := 0;
      timeUnit : UDInt := 1054;
   END_STRUCT;
END_TYPE

TYPE "SimaHydTO_typeHMIConnectionAxisToDataErrorDetail"
TITLE = SimaHydTO_typeHMIConnectionAxisToDataErrorDetail
// HMI interface: Technology object axis error detail
// stored: IsFailsafeCompliant false
   STRUCT
      number : UDInt;   // Error number
      reaction : DInt;   // Error reaction
   END_STRUCT;
END_TYPE

TYPE "SimaHydTO_typeHMIConnectionBasicAxisControl"
TITLE = SimaHydTO_typeHMIConnectionBasicAxisControl
// HMI interface: Basic axis control (LAxisBasics)
// stored: IsFailsafeCompliant false
   STRUCT
      Command { S7_SetPoint := 'True'} : "SimaHydTO_typeHMIConnectionBasicAxisControlCommand";
      Status { S7_SetPoint := 'True'} : "SimaHydTO_typeHMIConnectionBasicAxisControlStatus";
      ControlDirectOutput { S7_SetPoint := 'True'} : "SimaHydTO_typeIHMIConnectionBasicAxisControlDirectOutput";
      StatusDirectOutput { S7_SetPoint := 'True'} : "SimaHydTO_typeHMIConnectionBasicAxislStatusDirectOutput";
   END_STRUCT;
END_TYPE

TYPE "SimaHydTO_typeHMIConnectionBasicAxisControlCommand"
TITLE = SimaHydTO_typeHMIConnectionBasicAxisControlCommand
// HMI interface: Basic axis control (LAxisBasics) - Command (HMI -> PLC)
// stored: IsFailsafeCompliant false
   STRUCT
      powerEnable : Bool;   // MC_Power: 0: The technology object is disabled / 1: The technology object is enabled
      powerStartMode : DInt := 1;   // 0: Enable axis not position-controlled / 1: Enable axis position-controlled
      powerStopMode : Int := 0;   // 0: Emergency stop / 1: Immediate stop / 2: Stop with maximum dynamic values
      resetExecute : Bool;   // MC_Reset: Start job with a positive edge
      resetFBExecute : Bool;   // LSimaHyd_MC_Reset: Start job with a positive edge
      resetRestart : Bool := false;   // 0: Acknowledgment of queued technology alarms / 1: Reinitialization of the technology object and acknowledgment of pending technology alarms
      homeExecute : Bool;   // MC_Home: Start job with a positive edge
      homePosition : LReal;   // The specified value is used according to the selected "Mode".
      homeMode : Int;   // 0: Direct homing (absolute) / 1: Direct homing (relative) / 2: Passive homing / 3: Active homing / 4: Reserved / 5: Active homing (<TO>.Homing.HomePosition) / 6: Absolute encoder adjustment (relative) / 7: Absolute encoder adjustment (absolute) / 8: Passive homing / 9: Abort passive homing / 10: Passive homing (<TO>.Homing.HomePosition)
      jogForward : Bool;   // MC_MoveJog: As long as the parameter is TRUE, the axis moves in the positive direction
      jogBackward : Bool;   // MC_MoveJog: As long as the parameter is TRUE, the axis moves in the negative direction
      jogVelocity : LReal := 100.0;   // Velocity setpoint / speed setpoint for the motion
      jogAcceleration : LReal := -1.0;   // Acceleration of jog movement
      jogDeceleration : LReal := -1.0;   // Deceleration of jog movement
      jogJerk : LReal := -1.0;   // Jerk of jog movement
      jogPositionControlled : Bool := true;   // 0: Non position-controlled operation / 1: Position-controlled mode - The parameter applies as long as the MC_MoveJog command is executed. After this, the setting of MC_Power applies again.
   END_STRUCT;
END_TYPE

TYPE "SimaHydTO_typeHMIConnectionBasicAxisControlStatus"
TITLE = SimaHydTO_typeHMIConnectionBasicAxisControlStatus
// HMI interface: Basic axis control (LAxisBasics) - Status (PLC -> HMI)
// stored: IsFailsafeCompliant false
   STRUCT
      powerStatus : Bool;   // MC_Power: 0: Technology object disabled / 1: Technology object enabled
      powerBusy : Bool;   // MC_Power: Job is running
      resetDone : Bool;   // MC_Reset: Error has been acknowledged or Restart has been executed.
      resetBusy : Bool;   // MC_Reset: Job is running
      resetFBDone : Bool;   // LSimaHyd_MC_Reset: Error has been acknowledged or Restart has been executed.
      resetFBBusy : Bool;   // LSimaHyd_MC_Reset: Job is running
      homeDone : Bool;   // MC_Home: Job is completed
      homeBusy : Bool;   // MC_Home: Job is running
      jogInVelocity : Bool;   // MC_MoveJog: The velocity setpoint / speed setpoint was reached and will be maintained
      jogBusy : Bool;   // MC_MoveJog: Job is running
      commandAborted : Bool;   // The job was aborted by another job during execution (see also StatusID)
      error : Bool;   // An error occurred during execution of the job. The job is rejected. The cause of the error can be found in the "ErrorID" parameter.
      errorID : Word;   // ErrorID of motion control instruction (see also StatusID)
      statusID : Int;   // Additional specification of affected Motion control instruction of CommandAborted or Error: 0: No instruction / 1: MC_Power / 2: MC_Reset / 3: MC_Home / 4: MC_MoveJog
   END_STRUCT;
END_TYPE

TYPE "SimaHydTO_typeHMIConnectionBasicAxislStatusDirectOutput"
TITLE = SimaHydTO_typeHMIConnectionBasicAxislStatusDirectOutput
// Direct output status
// stored: IsFailsafeCompliant false
   STRUCT
      active : Bool;   // displays activity of direct output operation
      rampingDown : Bool;   // ramping down due to positioning limits
      minSafetyPositionOverrun : Bool;   // the min. safety position was passed
      maxSafetyPositionOverrun : Bool;   // the max. safety position was passed
   END_STRUCT;
END_TYPE

TYPE "SimaHydTO_typeHMIConnectionGetCharacteristicInterface"
TITLE = SimaHydTO_typeHMIConnectionGetCharacteristicInterface
// Function block interface of FB "GetCharacteristics"
// stored: IsFailsafeCompliant false
   STRUCT
      Command { S7_SetPoint := 'True'} : "SimaHydTO_typeHMIConnectionGetCharacteristicInterfaceCommand";   // HMI -> PLC: Commands to function block GetCharacteristics
      Status { S7_SetPoint := 'True'} : "SimaHydTO_typeHMIConnectionGetCharacteristicInterfaceStatus";   // PLC -> HMI: Status of function block GetCharacteristics
      ConfigData { S7_SetPoint := 'True'} : "LSimaHydTO_typeMeasurementConfig";
      MeasuredValues { S7_SetPoint := 'True'} : "LSimaHydTO_typeMeasuredValues";
   END_STRUCT;
END_TYPE

TYPE "SimaHydTO_typeHMIConnectionGetCharacteristicInterfaceCommand"
TITLE = SimaHydTO_typeHMIConnectionGetCharacteristicInterfaceCommand
// Function block command interface of FB "GetCharacteristics"
// stored: IsFailsafeCompliant false
   STRUCT
      execute : Bool;   // Start measurement
      abort : Bool;   // Stop measurement
      enableRampingForward : Bool := True;   // Enable ramping of Q-Output value (voltage) in positivedirection
      enableRampingBackward : Bool := True;   // Enable ramping of Q-Output value (voltage) in negative direction
      saveConfig : Bool;   // Save measurement configuration
      loadConfig : Bool;   // Load measurement configuration
   END_STRUCT;
END_TYPE

TYPE "SimaHydTO_typeHMIConnectionGetCharacteristicInterfaceStatus"
TITLE = SimaHydTO_typeHMIConnectionGetCharacteristicInterfaceStatus
// Function block status interface of FB "GetCharacteristics"
// stored: IsFailsafeCompliant false
   STRUCT
      qOutputValueStepForward { ExternalWritable := 'False'} : LReal;   // Last successfully measured manipulated variable in the positive direction
      qOutputValueStepBackward { ExternalWritable := 'False'} : LReal;   // Last successfully measured velocity in the negative direction
      velocityStepForward { ExternalWritable := 'False'} : LReal;   // Last successfully measured velocity in the positive direction
      velocityStepBackward { ExternalWritable := 'False'} : LReal;   // Last successfully measured velocity in the negative direction
      requestForward { ExternalWritable := 'False'} : Bool;   // Request switching to move in the positive direction
      requestBackward { ExternalWritable := 'False'} : Bool;   // Request switching to move in the negative direction
      statusMeasurement { ExternalWritable := 'False'} : Word;   // Status of current measurement
      done { ExternalWritable := 'False'} : Bool;   // The measurement was successfully completed
      busy { ExternalWritable := 'False'} : Bool;   // Measurement active
      commandAborted { ExternalWritable := 'False'} : Bool;   // Measurement function was interrupted
      error { ExternalWritable := 'False'} : Bool;   // There is an error in the FB
      status { ExternalWritable := 'False'} : Word;   // Error information or status of the block
   END_STRUCT;
END_TYPE

TYPE "SimaHydTO_typeHMIConnectionHmiData"
TITLE = SimaHydTO_typeHMIConnectionHmiData
// HMI interface: Data to display on HMI
// stored: IsFailsafeCompliant false
   STRUCT
      stateSubNavigation : Int;
      ActualPositionPercent : Int;   // Actual axis position in percent between MinPosition and MaxPosition
      SafetyDistanceAnimation : LReal;   // SafetyDistance in percent between MinPosition and MaxPosition
      MinPosition : LReal;   // Minimal position of axis (SW limit switch)
      MaxPosition : LReal;   // Maximal position of axis (SW limit switch)
      selectedAxis : Int;   // DB number of actual selected hydraulic axis
      selectedAxisTO : Int;   // DB/TO number of actual selected technology object
      selectedVChar : Int;   // DB number of actual selected valve characteristics
      VChar { S7_SetPoint := 'True'} : "SimaHydTO_typeHMIConnectionHmiDataVChar";   // Data storage of HMI VChar display
   END_STRUCT;
END_TYPE

TYPE "SimaHydTO_typeHMIConnectionHmiDataVChar"
TITLE = SimaHydTO_typeHMIConnectionHmiDataVChar
// HMI interface: Calculated positions of VHar to display on HMI
// stored: IsFailsafeCompliant false
   STRUCT
      HMI_VChar : Array[1..200] of Real;
      HMI_VChar_MinQOutput : Real;
      HMI_VChar_MaxQOutput : Real;
      HMI_VChar_MinVelocity : Real;
      HMI_VCHar_MaxVelocity : Real;
      HMI_VChar_TrendRequest : Word;
      HMI_VChar_TrendTransfer : Word;
   END_STRUCT;
END_TYPE

TYPE "SimaHydTO_typeHMIConnectionParameterSettings"
TITLE = SimaHydTO_typeHMIConnectionParameterSettings
// HMI interface: Parameter settings
// stored: IsFailsafeCompliant false
   STRUCT
      AxisData { S7_SetPoint := 'True'} : "SimaHydTO_typeHMIConnectionParameterSettingsAxisData";
      Commands { S7_SetPoint := 'True'} : "SimaHydTO_typeHMIConnectionParameterSettingsCommands";   // Data: HMI -> PLC
      Status { S7_SetPoint := 'True'} : "SimaHydTO_typeHMIConnectionParameterSettingsStatus";   // Data: PLC -> HMI
   END_STRUCT;
END_TYPE

TYPE "SimaHydTO_typeHMIConnectionParameterSettingsAxisData"
TITLE = SimaHydTO_typeHMIConnectionParameterSettingsAxisData
// Axis data
// stored: IsFailsafeCompliant false
   STRUCT
      Actor { S7_SetPoint := 'True'} : "LSimaHydTO_typeActor";   // Actor configuration
      ValveCharacteristic { S7_SetPoint := 'True'} : "LSimaHydTO_typeValveCharacteristic";   // Valve characteristic
      ForceLimits { S7_SetPoint := 'True'} : "LSimaHydTO_typeForceLimits";   // Force limits
      Pressure_A_Transducer { S7_SetPoint := 'True'} : "LSimaHydTO_typeTransducer";   // Piston side pressure transducer configuration
      Pressure_B_Transducer { S7_SetPoint := 'True'} : "LSimaHydTO_typeTransducer";   // Piston rod side pressure transducer configuration
      PositionControl { S7_SetPoint := 'True'} : "LSimaHydTO_typePositionControl";   // Position control configuration data
      ForceControl { S7_SetPoint := 'True'} : "LSimaHydTO_typeForceControl";   // Force control configuration data
      DynamicAxisModel { S7_SetPoint := 'True'} : "LSimaHydTO_typeDynamicAxisModel";   // Settings of the balancing filter
      SmoothingFilter { S7_SetPoint := 'True'} : "LSimaHydTO_typeSmoothingFilter";   // Settings of the smoothing filter
      StatusActor { S7_SetPoint := 'True'} : "LSimaHydTO_typeStatusActor";   // Indicates the status of actor data
      StatusVChar { S7_SetPoint := 'True'} : "LSimaHydTO_typeStatusVChar";   // Indicates the status of valve characteristic data
      Status_A_Transducer { S7_SetPoint := 'True'} : "LSimaHydTO_typeStatusTransducer";   // Indicates the status of piston side pressure transducer data
      Status_B_Transducer { S7_SetPoint := 'True'} : "LSimaHydTO_typeStatusTransducer";   // Indicates the status of piston rod side pressure transducer data
      StatusServo { S7_SetPoint := 'True'} : "LSimaHydTO_typeStatusServo";   // Indicates the status of position control
      StatusForce { S7_SetPoint := 'True'} : "LSimaHydTO_typeStatusForce";   // Indicates the status of force control
      StatusForceProfile { S7_SetPoint := 'True'} : "LSimaHydTO_typeStatusForceProfile";   // Indicates the status of a force profile processing
      "Name" : WString[24];   // Name displayed on HMI
      VCharName : WString[24];   // Charachteristic name displayed on HMI
   END_STRUCT;
END_TYPE

TYPE "SimaHydTO_typeHMIConnectionParameterSettingsCommands"
TITLE = SimaHydTO_typeHMIConnectionParameterSettingsCommands
// HMI interface: Parameter settings - Command (HMI -> PLC)
// stored: IsFailsafeCompliant false
   STRUCT
      Edit : Bool;
      Activate : Bool;
      Save : Bool;
      Restore : Bool;
      Abort : Bool;
      ApplyVChar : Bool;
      VCharSelector { S7_SetPoint := 'True'} : "SimaHydTO_typeHMIConnectionVCharSelectorCommand";
   END_STRUCT;
END_TYPE

TYPE "SimaHydTO_typeHMIConnectionParameterSettingsStatus"
TITLE = SimaHydTO_typeHMIConnectionParameterSettingsStatus
// HMI interface: Parameter settings - Status (PLC -> HMI)
// stored: IsFailsafeCompliant false
   STRUCT
      EditorActive : Bool;
      StateActivation : Int;   // 0: none / 1: activated / 2: error
      StateSaving : Int;   // 0: none / 1: saved / 2: error
      StateLoading : Int;   // 0: none / 1: restoreded / 2: error
      VCharSelector { S7_SetPoint := 'True'} : "SimaHydTO_typeHMIConnectionVCharSelectorStatus";
   END_STRUCT;
END_TYPE

TYPE "SimaHydTO_typeHMIConnectionVCharEditor"
TITLE = SimaHydTO_typeHMIConnectionVCharEditor
// HMI interface: VChar editor
// stored: IsFailsafeCompliant false
   STRUCT
      Command { S7_SetPoint := 'True'} : "SimaHydTO_typeHMIConnectionVCharEditorCommand";   // Data: HMI -> PLC
      Status { S7_SetPoint := 'True'} : "SimaHydTO_typeHMIConnectionVCharEditorStatus";   // Data: PLC -> HMI
      Parameter { S7_SetPoint := 'True'} : "SimaHydTO_typeHMIConnectionVCharEditorParameter";   // Data: PLC <-> HMI (Load and save)
      Table { S7_SetPoint := 'True'} : "SimaHydTO_typeHMIConnectionVCharEditorTable";   // Data table of VChar
      VCharNameToSave : WString[24];   // Name of VChar to be saved
   END_STRUCT;
END_TYPE

TYPE "SimaHydTO_typeHMIConnectionVCharEditorCommand"
TITLE = SimaHydTO_typeHMIConnectionVCharEditorCommand
// HMI interface: VChar editor - Command (HMI -> PLC)
// stored: IsFailsafeCompliant false
   STRUCT
      LoadMeasuredValues : Bool;
      LoadVChar : Bool;
      VCharLoad { S7_SetPoint := 'True'} : "SimaHydTO_typeHMIConnectionVCharSelectorCommand";
      CreateNewVChar : Bool;
      ShowPreviousRow : Bool;
      ShowNextRow : Bool;
      SaveVChar : Bool;
      SaveVCharAs : Bool;
      VCharSave { S7_SetPoint := 'True'} : "SimaHydTO_typeHMIConnectionVCharSelectorCommand";
      AbortEditor : Bool;
      DeleteRow : Bool;
      AddRow : Bool;
      SortAndDisplay : Bool;
   END_STRUCT;
END_TYPE

TYPE "SimaHydTO_typeHMIConnectionVCharEditorParameter"
TITLE = SimaHydTO_typeHMIConnectionVCharEditorParameter
// HMI interface: VChar editor
// stored: IsFailsafeCompliant false
   STRUCT
      ActualTableStartIndex : Int;
      SelectedTableIndex : Int;
      MaximumNumberOfLines : Int;
      NumberOfUsedLines : Int;
      NumberOfUsableLines : Int;
   END_STRUCT;
END_TYPE

TYPE "SimaHydTO_typeHMIConnectionVCharEditorStatus"
TITLE = SimaHydTO_typeHMIConnectionVCharEditorStatus
// HMI interface: VChar editor - Status (PLC -> HMI)
// stored: IsFailsafeCompliant false
   STRUCT
      EditorActive : Bool;
      SaveAsSelected : Bool;
      Busy : Bool;
      Error : Bool;
      VCharLoad { S7_SetPoint := 'True'} : "SimaHydTO_typeHMIConnectionVCharSelectorStatus";
      VCharSave { S7_SetPoint := 'True'} : "SimaHydTO_typeHMIConnectionVCharSelectorStatus";
   END_STRUCT;
END_TYPE

TYPE "SimaHydTO_typeHMIConnectionVCharEditorTable"
TITLE = SimaHydTO_typeHMIConnectionVCharEditorTable
// HMI interface: VChar editor
// stored: IsFailsafeCompliant false
   STRUCT
      Appearance : Array[0..20] of Int;   // 0: invisible / 1: visible / 2: selected
      Index : Array[0..20] of Int;
      Velocity : Array[0..20] of Real;
      QOutput : Array[0..20] of Real;
      VelocityLimitPositive : Real;   // Max velocity in positive direction
      VelocityLimitNegative : Real;   // Max velocity in negative direction
      ZeroZonePositive : Real;   // Overlapping zone of valve in positive direction
      ZeroZoneNegative : Real;   // Overlapping zone of valve in negative direction
   END_STRUCT;
END_TYPE

TYPE "SimaHydTO_typeHMIConnectionVCharSelectorCommand"
TITLE = SimaHydTO_typeHMIConnectionVCharSelectorCommand
// HMI interface: Hydraulic characteristics (VChar) selection of VChar array - Command (HMI -> PLC)
// stored: IsFailsafeCompliant false
   STRUCT
      previousObject : Bool;
      nextObject : Bool;
      executeDirectIndexSelection : Bool;
      directIndexSelection : Int;
   END_STRUCT;
END_TYPE

TYPE "SimaHydTO_typeHMIConnectionVCharSelectorStatus"
TITLE = SimaHydTO_typeHMIConnectionVCharSelectorStatus
// HMI interface: Hydraulic characteristics (VChar) selection of VChar array - Status (PLC -> HMI)
// stored: IsFailsafeCompliant false
   STRUCT
      actualVCharIndex : Int;   // Actual selected array index
      selectedVCharInteger : UInt;   // DB number of actual selected valve characteristics as integer value
      selectedVChar : DB_ANY;   // DB number of actual selected valve characteristics
      selectedVCharName : WString[24];   // Name of actual selected valve characteristics
      dataValid : Bool;   // Selected data valid
      dataError : Bool;   // Error of data selection
   END_STRUCT;
END_TYPE

TYPE "SimaHydTO_typeIHMIConnectionBasicAxisControlDirectOutput"
TITLE = SimaHydTO_typeIHMIConnectionBasicAxisControlDirectOutput
// Direct output control
// stored: IsFailsafeCompliant false
   STRUCT
      jogForward : Bool;   // Direct output is active in positive direction if TRUE
      jogBackward : Bool;   // Direct output is active in negative direction if TRUE
      commandValueForward : LReal := 5.0;   // Direct output value in positive direction [%]
      commandValueBackward : LReal := 5.0;   // Direct output value in negative direction [%]
      commandValueRamp : LReal := 100.0;   // Ramp for command value [%/s]
      safetyDistance : LReal := 50.0;   // Safety distance to avoid passing over the min. and max. positions
   END_STRUCT;
END_TYPE

TYPE "SimaHydTO_typeVCharArray"
TITLE = SimaHydTO_typeVCharArray
// VChar (characteristics) array of HMI VChar selection
// stored: IsFailsafeCompliant false
   STRUCT
      VChar_DB : DB_ANY;   // DB number of VChar storage
      measurementConfig { S7_SetPoint := 'True'} : "LSimaHydTO_typeMeasurementConfig";
      initialized : Bool;
   END_STRUCT;
END_TYPE

DATA_BLOCK "DENEME"   // DB3
{ S7_Optimized_Access := 'TRUE' }
VERSION : 0.1
// stored: AutoNumber true, DBAccessibleFromOPCUA true, IsOnlyStoredInLoadMemory false, IsRetainMemResEnabled false, IsWriteProtectedInAS false, MemoryReserve 100
   VAR
      VELO : Real;
      RESET : Bool;
      MoveABS : Bool;
      AbsolutePoz : Real;
      ABSvelo : Real;
      CETVEL : Real;
      HOME : Bool;
      ABSOLUTE_AUX : Real;
      OFFSET : Real;
   END_VAR
BEGIN
END_DATA_BLOCK

DATA_BLOCK "HydAxisAnalogInterface1"   // DB33150
{ S7_Optimized_Access := 'TRUE' }
FAMILY : SimaHydTO
VERSION : 1.0
// stored: AutoNumber true, DBAccessibleFromOPCUA true, IsOnlyStoredInLoadMemory false, IsRetainMemResEnabled false, IsWriteProtectedInAS false, MemoryReserve 0
   VAR
      tel81 { ExternalAccessible := 'False'; ExternalVisible := 'False'; ExternalWritable := 'False'; S7_SetPoint := 'True'} : PD_TEL81;
   END_VAR
BEGIN
END_DATA_BLOCK

DATA_BLOCK "HydAxisAnalogInterface2"   // DB33151
{ S7_Optimized_Access := 'TRUE' }
FAMILY : SimaHydTO
VERSION : 1.0
// stored: AutoNumber true, DBAccessibleFromOPCUA true, IsOnlyStoredInLoadMemory false, IsRetainMemResEnabled false, IsWriteProtectedInAS false, MemoryReserve 0
   VAR
      tel81 { ExternalAccessible := 'False'; ExternalVisible := 'False'; ExternalWritable := 'False'; S7_SetPoint := 'True'} : PD_TEL81;
   END_VAR
BEGIN
END_DATA_BLOCK

DATA_BLOCK "HydAxisDriveInterface"   // DB33152
{ S7_Optimized_Access := 'FALSE'; DB_Accessible_From_OPC_UA := 'FALSE' }
FAMILY : SimaHydTO
VERSION : 1.0
// stored: AutoNumber true, DBAccessibleFromOPCUA false, IsOnlyStoredInLoadMemory false, IsWriteProtectedInAS false
   VAR
      tel2 { ExternalAccessible := 'False'; ExternalVisible := 'False'; ExternalWritable := 'False'; S7_SetPoint := 'True'} : PD_TEL2;
      tel81 { ExternalAccessible := 'False'; ExternalVisible := 'False'; ExternalWritable := 'False'; S7_SetPoint := 'True'} : PD_TEL81;
   END_VAR
BEGIN
END_DATA_BLOCK

DATA_BLOCK "LSimaHydTO_HydAxisAnalogInterfaceTemplate"   // DB33050
TITLE = LSimaHydTO_HydAxisAnalogInterfaceTemplate
{ S7_Optimized_Access := 'TRUE'; DB_Accessible_From_OPC_UA := 'FALSE' }
AUTHOR : APC_ERLF
FAMILY : LSimaHydTO
VERSION : 1.0
// stored: AutoNumber true, DBAccessibleFromOPCUA false, IsOnlyStoredInLoadMemory false, IsRetainMemResEnabled false, IsWriteProtectedInAS false, MemoryReserve 0
   VAR
      tel81 { ExternalAccessible := 'False'; ExternalVisible := 'False'; ExternalWritable := 'False'; S7_SetPoint := 'True'} : PD_TEL81;
   END_VAR
BEGIN
END_DATA_BLOCK

DATA_BLOCK "LSimaHydTO_HydAxisDriveInterfaceTemplate"   // DB33051
TITLE = LSimaHydTO_HydAxisDriveInterfaceTemplate
{ S7_Optimized_Access := 'FALSE'; DB_Accessible_From_OPC_UA := 'FALSE' }
AUTHOR : APC_ERLF
FAMILY : LSimaHydTO
VERSION : 1.0
// stored: AutoNumber true, DBAccessibleFromOPCUA false, IsOnlyStoredInLoadMemory false, IsWriteProtectedInAS false
   VAR
      tel2 { ExternalAccessible := 'False'; ExternalVisible := 'False'; ExternalWritable := 'False'; S7_SetPoint := 'True'} : PD_TEL2;
      tel81 { ExternalAccessible := 'False'; ExternalVisible := 'False'; ExternalWritable := 'False'; S7_SetPoint := 'True'} : PD_TEL81;
   END_VAR
BEGIN
END_DATA_BLOCK

DATA_BLOCK "SimaHydTO_AxesArray"   // DB33101
TITLE = SimaHydTO_AxesArray
{ S7_Optimized_Access := 'TRUE'; DB_Accessible_From_OPC_UA := 'FALSE' }
FAMILY : SimaHydTO
VERSION : 1.0
// Array of hydraulic axes usabel in HMI
// stored: AutoNumber true, DBAccessibleFromOPCUA false, IsOnlyStoredInLoadMemory false, IsRetainMemResEnabled false, IsWriteProtectedInAS false, MemoryReserve 100
   VAR
      axes { S7_SetPoint := 'True'} : Array[0..2] of "SimaHydTO_typeAxesArray";   // Hydraulic axes of the project to be controlled via HMI
   END_VAR
BEGIN
END_DATA_BLOCK

DATA_BLOCK "SimaHydTO_VCharArray"   // DB33102
TITLE = SimaHydTO_VCharArray
{ S7_Optimized_Access := 'TRUE'; DB_Accessible_From_OPC_UA := 'FALSE' }
FAMILY : SimaHydTO
VERSION : 1.0
// Array of valve chracteristics usabel in HMI
// stored: AutoNumber true, DBAccessibleFromOPCUA false, IsOnlyStoredInLoadMemory false, IsRetainMemResEnabled false, IsWriteProtectedInAS false, MemoryReserve 100
   VAR
      VChar { S7_SetPoint := 'True'} : Array[0..12] of "SimaHydTO_typeVCharArray";   // Valve charactersitics of the project to be controlled via HMI
   END_VAR
BEGIN
   VChar[0].VChar_DB := 5001;
END_DATA_BLOCK

ORGANIZATION_BLOCK "Main"   // OB1, FBD, ProgramCycle
TITLE = "Main Program Sweep (Cycle)"
{ S7_Optimized_Access := 'TRUE' }
VERSION : 0.1
// stored: AutoNumber true, IsIECCheckEnabled false, SetENOAutomatically false
   VAR_INPUT
      Initial_Call : Bool;   // Initial call of this OB
      Remanence : Bool;   // =True, if remanent data are available
   END_VAR
BEGIN
END_ORGANIZATION_BLOCK

ORGANIZATION_BLOCK "MC-PostServo"   // OB95, LAD, PostServo
{ S7_Optimized_Access := 'TRUE' }
VERSION : 0.1
// stored: IsIECCheckEnabled false, SetENOAutomatically false
   VAR_INPUT
      Initial_Call : Bool;
      PIP_Input : Bool;
      PIP_Output : Bool;
      IO_System : USInt;
      Event_Count : Int;
      Synchronous : Bool;
      CycleTime : UDInt;
   END_VAR
   VAR_TEMP
      tempCycleTime : LReal;
      tempCycleTimeLINT : LInt;
      tempRetVal : Word;
      VELOO : Real;
      cetvel2 : Real;
   END_VAR
   VAR_TEMP   // added for the SCL form of the ladder/FBD networks
      _w1 : Bool;
      _w2 : Bool;
   END_VAR
BEGIN

REGION Network 1: Set characteristics of axis at first call
   // Initial setting of valve characteristics.
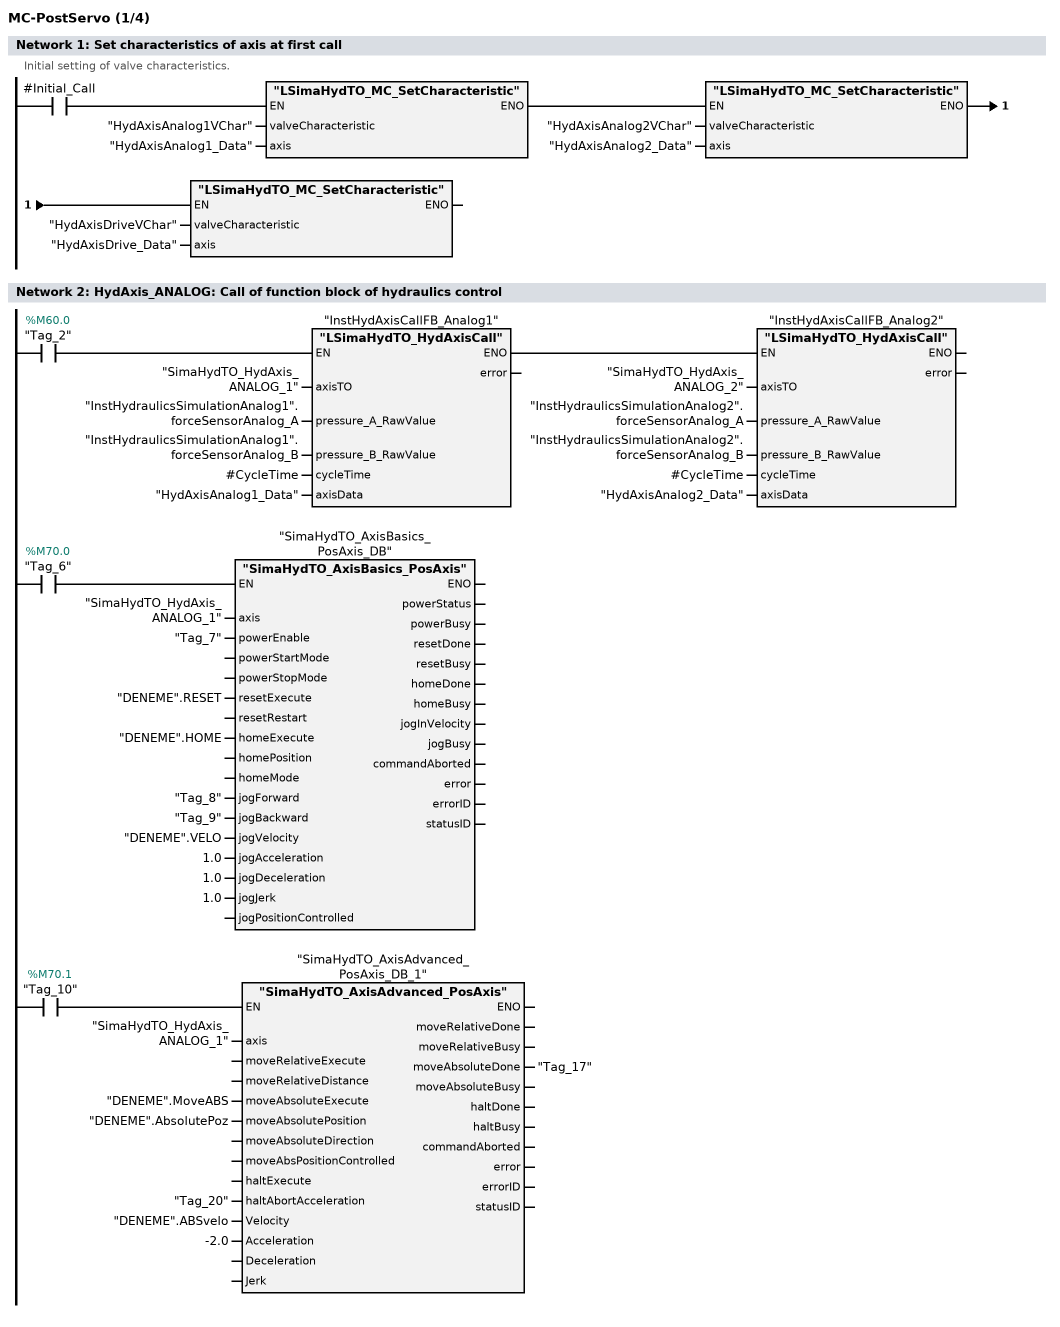
   RUNG wire#powerrail
      Contact( #Initial_Call )
      "LSimaHydTO_MC_SetCharacteristic"(valveCharacteristic := "HydAxisAnalog1VChar", axis := "HydAxisAnalog1_Data")
      "LSimaHydTO_MC_SetCharacteristic"(valveCharacteristic := "HydAxisAnalog2VChar", axis := "HydAxisAnalog2_Data")
      "LSimaHydTO_MC_SetCharacteristic"(valveCharacteristic := "HydAxisDriveVChar", axis := "HydAxisDrive_Data")
   END_RUNG
   // the same network as SCL:
   "LSimaHydTO_MC_SetCharacteristic"(EN := #Initial_Call,
                           valveCharacteristic := "HydAxisAnalog1VChar",
                           axis := "HydAxisAnalog1_Data",
                           ENO => #_w1);
   "LSimaHydTO_MC_SetCharacteristic"(EN := #_w1,
                           valveCharacteristic := "HydAxisAnalog2VChar",
                           axis := "HydAxisAnalog2_Data",
                           ENO => #_w2);
   IF #_w2 THEN
       "LSimaHydTO_MC_SetCharacteristic"(valveCharacteristic := "HydAxisDriveVChar", axis := "HydAxisDrive_Data");
   END_IF;
END_REGION

REGION Network 2: HydAxis_ANALOG: Call of function block of hydraulics control
   RUNG wire#powerrail
      Contact( "Tag_2" )
      "InstHydAxisCallFB_Analog1"(axisTO := "SimaHydTO_HydAxis_ANALOG_1", pressure_A_RawValue := "InstHydraulicsSimulationAnalog1".forceSensorAnalog_A, pressure_B_RawValue := "InstHydraulicsSimulationAnalog1".forceSensorAnalog_B, cycleTime := #CycleTime, axisData := "HydAxisAnalog1_Data", error =>)
      "InstHydAxisCallFB_Analog2"(axisTO := "SimaHydTO_HydAxis_ANALOG_2", pressure_A_RawValue := "InstHydraulicsSimulationAnalog2".forceSensorAnalog_A, pressure_B_RawValue := "InstHydraulicsSimulationAnalog2".forceSensorAnalog_B, cycleTime := #CycleTime, axisData := "HydAxisAnalog2_Data", error =>)
   END_RUNG
   RUNG wire#powerrail
      Contact( "Tag_6" )
      "SimaHydTO_AxisBasics_PosAxis_DB"(axis := "SimaHydTO_HydAxis_ANALOG_1", powerEnable := "Tag_7", powerStartMode :=, powerStopMode :=, resetExecute := "DENEME".RESET, resetRestart :=, homeExecute := "DENEME".HOME, homePosition :=, homeMode :=, jogForward := "Tag_8", jogBackward := "Tag_9", jogVelocity := "DENEME".VELO, jogAcceleration := 1.0, jogDeceleration := 1.0, jogJerk := 1.0, jogPositionControlled :=, powerStatus =>, powerBusy =>, resetDone =>, resetBusy =>, homeDone =>, homeBusy =>, jogInVelocity =>, jogBusy =>, commandAborted =>, error =>, errorID =>, statusID =>)
   END_RUNG
   RUNG wire#powerrail
      Contact( "Tag_10" )
      "SimaHydTO_AxisAdvanced_PosAxis_DB_1"(axis := "SimaHydTO_HydAxis_ANALOG_1", moveRelativeExecute :=, moveRelativeDistance :=, moveAbsoluteExecute := "DENEME".MoveABS, moveAbsolutePosition := "DENEME".AbsolutePoz, moveAbsoluteDirection :=, moveAbsPositionControlled :=, haltExecute :=, haltAbortAcceleration := "Tag_20", Velocity := "DENEME".ABSvelo, Acceleration := -2.0, Deceleration :=, Jerk :=, moveRelativeDone =>, moveRelativeBusy =>, moveAbsoluteDone => "Tag_17", moveAbsoluteBusy =>, haltDone =>, haltBusy =>, commandAborted =>, error =>, errorID =>, statusID =>)
   END_RUNG
   // the same network as SCL:
   "InstHydAxisCallFB_Analog1"(EN := "Tag_2",   // "LSimaHydTO_HydAxisCall"
                           axisTO := "SimaHydTO_HydAxis_ANALOG_1",
                           pressure_A_RawValue := "InstHydraulicsSimulationAnalog1".forceSensorAnalog_A,
                           pressure_B_RawValue := "InstHydraulicsSimulationAnalog1".forceSensorAnalog_B,
                           cycleTime := #CycleTime,
                           axisData := "HydAxisAnalog1_Data",
                           ENO => #_w1);
   IF #_w1 THEN
       "InstHydAxisCallFB_Analog2"(axisTO := "SimaHydTO_HydAxis_ANALOG_2",   // "LSimaHydTO_HydAxisCall"
                               pressure_A_RawValue := "InstHydraulicsSimulationAnalog2".forceSensorAnalog_A,
                               pressure_B_RawValue := "InstHydraulicsSimulationAnalog2".forceSensorAnalog_B,
                               cycleTime := #CycleTime,
                               axisData := "HydAxisAnalog2_Data");
   END_IF;
   IF "Tag_6" THEN
       "SimaHydTO_AxisBasics_PosAxis_DB"(axis := "SimaHydTO_HydAxis_ANALOG_1",   // "SimaHydTO_AxisBasics_PosAxis"
                               powerEnable := "Tag_7",
                               resetExecute := "DENEME".RESET,
                               homeExecute := "DENEME".HOME,
                               jogForward := "Tag_8",
                               jogBackward := "Tag_9",
                               jogVelocity := "DENEME".VELO,
                               jogAcceleration := 1.0,
                               jogDeceleration := 1.0,
                               jogJerk := 1.0);
   END_IF;
   IF "Tag_10" THEN
       "SimaHydTO_AxisAdvanced_PosAxis_DB_1"(axis := "SimaHydTO_HydAxis_ANALOG_1",   // "SimaHydTO_AxisAdvanced_PosAxis"
                               moveAbsoluteExecute := "DENEME".MoveABS,
                               moveAbsolutePosition := "DENEME".AbsolutePoz,
                               haltAbortAcceleration := "Tag_20",
                               Velocity := "DENEME".ABSvelo,
                               Acceleration := -2.0,
                               moveAbsoluteDone => "Tag_17");
   END_IF;
END_REGION

REGION Network 3: HydAxis_ANALOG: Call of function block of hydraulics axis simulation
   // The simulation uses as input signal "analogInput" the real output integer value of analog module AQ. (-27648...+27648)
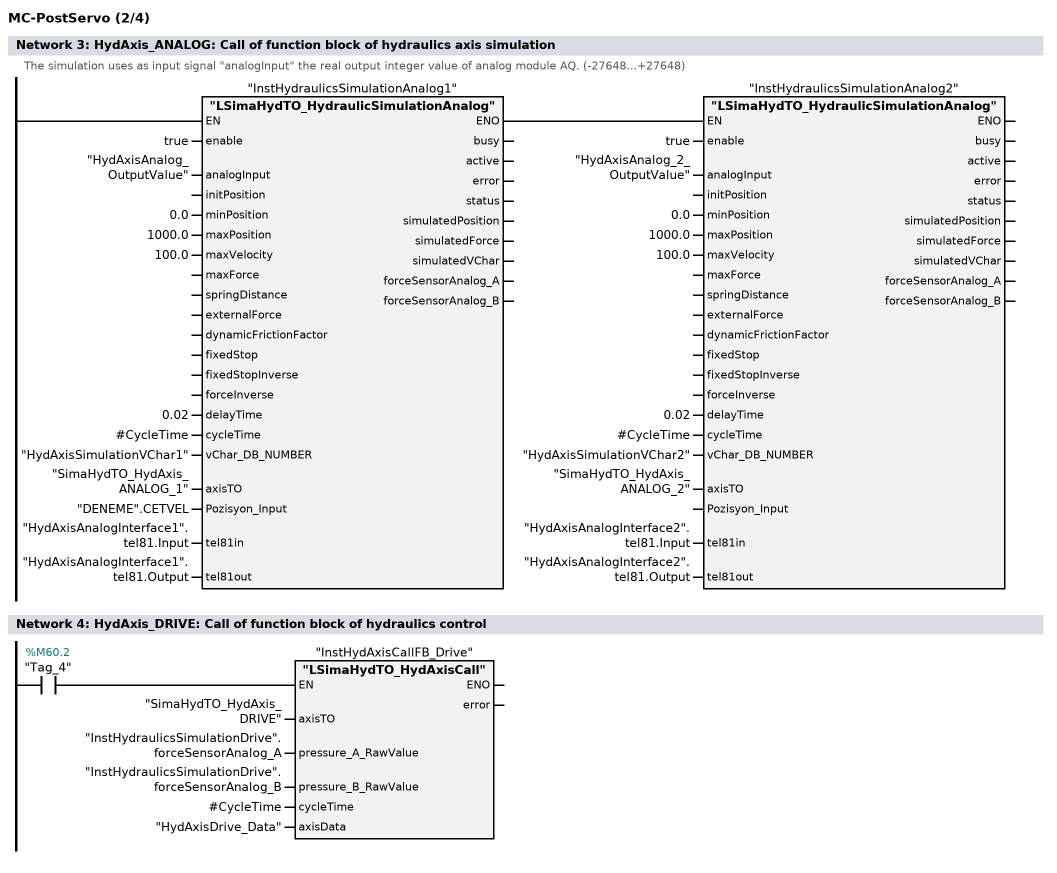
   RUNG wire#powerrail
      "InstHydraulicsSimulationAnalog1"(enable := true, analogInput := "HydAxisAnalog_OutputValue", initPosition :=, minPosition := 0.0, maxPosition := 1000.0, maxVelocity := 100.0, maxForce :=, springDistance :=, externalForce :=, dynamicFrictionFactor :=, fixedStop :=, fixedStopInverse :=, forceInverse :=, delayTime := 0.02, cycleTime := #CycleTime, vChar_DB_NUMBER := "HydAxisSimulationVChar1", axisTO := "SimaHydTO_HydAxis_ANALOG_1", Pozisyon_Input := "DENEME".CETVEL, tel81in := "HydAxisAnalogInterface1".tel81.Input, tel81out := "HydAxisAnalogInterface1".tel81.Output, busy =>, active =>, error =>, status =>, simulatedPosition =>, simulatedForce =>, simulatedVChar =>, forceSensorAnalog_A =>, forceSensorAnalog_B =>)
      "InstHydraulicsSimulationAnalog2"(enable := true, analogInput := "HydAxisAnalog_2_OutputValue", initPosition :=, minPosition := 0.0, maxPosition := 1000.0, maxVelocity := 100.0, maxForce :=, springDistance :=, externalForce :=, dynamicFrictionFactor :=, fixedStop :=, fixedStopInverse :=, forceInverse :=, delayTime := 0.02, cycleTime := #CycleTime, vChar_DB_NUMBER := "HydAxisSimulationVChar2", axisTO := "SimaHydTO_HydAxis_ANALOG_2", Pozisyon_Input :=, tel81in := "HydAxisAnalogInterface2".tel81.Input, tel81out := "HydAxisAnalogInterface2".tel81.Output, busy =>, active =>, error =>, status =>, simulatedPosition =>, simulatedForce =>, simulatedVChar =>, forceSensorAnalog_A =>, forceSensorAnalog_B =>)
   END_RUNG
   // the same network as SCL:
   "InstHydraulicsSimulationAnalog1"(enable := true,   // "LSimaHydTO_HydraulicSimulationAnalog"
                           analogInput := "HydAxisAnalog_OutputValue",
                           minPosition := 0.0,
                           maxPosition := 1000.0,
                           maxVelocity := 100.0,
                           delayTime := 0.02,
                           cycleTime := #CycleTime,
                           vChar_DB_NUMBER := "HydAxisSimulationVChar1",
                           axisTO := "SimaHydTO_HydAxis_ANALOG_1",
                           Pozisyon_Input := "DENEME".CETVEL,
                           tel81in := "HydAxisAnalogInterface1".tel81.Input,
                           tel81out := "HydAxisAnalogInterface1".tel81.Output,
                           ENO => #_w1);
   IF #_w1 THEN
       "InstHydraulicsSimulationAnalog2"(enable := true,   // "LSimaHydTO_HydraulicSimulationAnalog"
                               analogInput := "HydAxisAnalog_2_OutputValue",
                               minPosition := 0.0,
                               maxPosition := 1000.0,
                               maxVelocity := 100.0,
                               delayTime := 0.02,
                               cycleTime := #CycleTime,
                               vChar_DB_NUMBER := "HydAxisSimulationVChar2",
                               axisTO := "SimaHydTO_HydAxis_ANALOG_2",
                               tel81in := "HydAxisAnalogInterface2".tel81.Input,
                               tel81out := "HydAxisAnalogInterface2".tel81.Output);
   END_IF;
END_REGION

REGION Network 4: HydAxis_DRIVE: Call of function block of hydraulics control
   RUNG wire#powerrail
      Contact( "Tag_4" )
      "InstHydAxisCallFB_Drive"(axisTO := "SimaHydTO_HydAxis_DRIVE", pressure_A_RawValue := "InstHydraulicsSimulationDrive".forceSensorAnalog_A, pressure_B_RawValue := "InstHydraulicsSimulationDrive".forceSensorAnalog_B, cycleTime := #CycleTime, axisData := "HydAxisDrive_Data", error =>)
   END_RUNG
   // the same network as SCL:
   IF "Tag_4" THEN
       "InstHydAxisCallFB_Drive"(axisTO := "SimaHydTO_HydAxis_DRIVE",   // "LSimaHydTO_HydAxisCall"
                               pressure_A_RawValue := "InstHydraulicsSimulationDrive".forceSensorAnalog_A,
                               pressure_B_RawValue := "InstHydraulicsSimulationDrive".forceSensorAnalog_B,
                               cycleTime := #CycleTime,
                               axisData := "HydAxisDrive_Data");
   END_IF;
END_REGION

REGION Network 5: HydAxis_DRIVE: Call of function block of hydraulics axis simulation
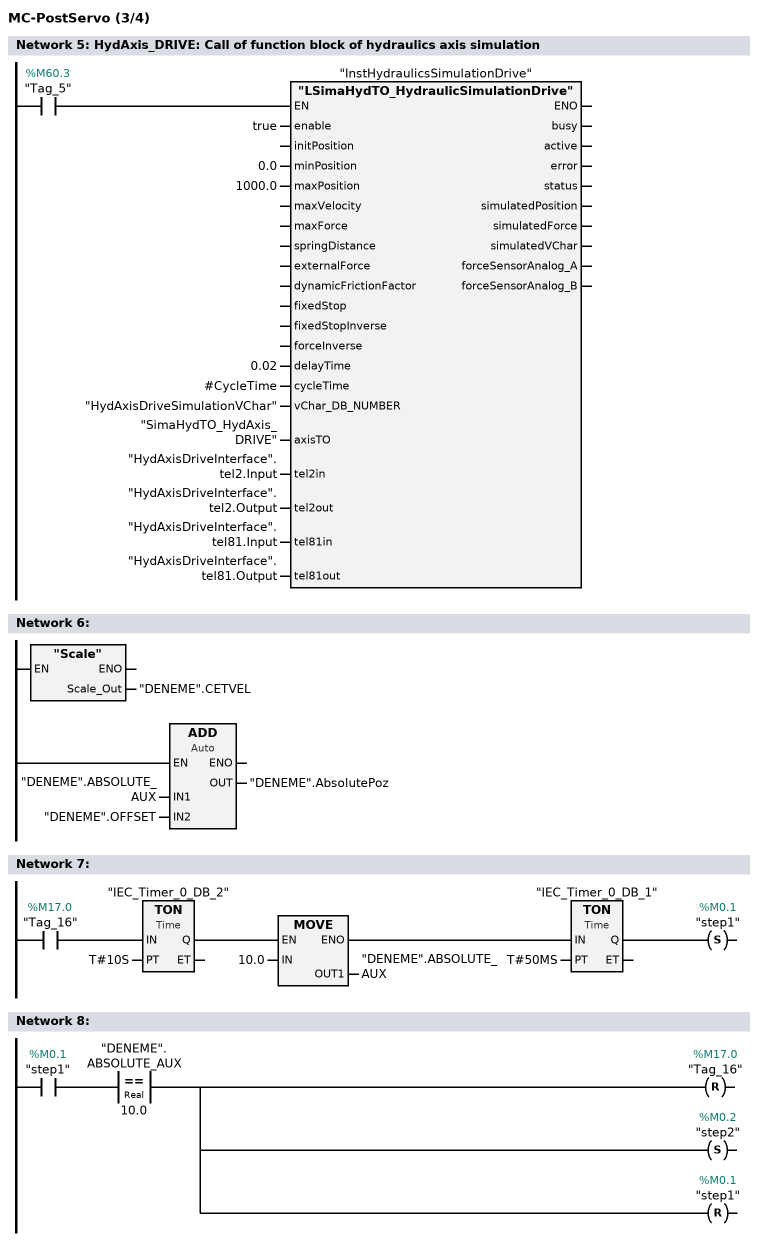
   RUNG wire#powerrail
      Contact( "Tag_5" )
      "InstHydraulicsSimulationDrive"(enable := true, initPosition :=, minPosition := 0.0, maxPosition := 1000.0, maxVelocity :=, maxForce :=, springDistance :=, externalForce :=, dynamicFrictionFactor :=, fixedStop :=, fixedStopInverse :=, forceInverse :=, delayTime := 0.02, cycleTime := #CycleTime, vChar_DB_NUMBER := "HydAxisDriveSimulationVChar", axisTO := "SimaHydTO_HydAxis_DRIVE", tel2in := "HydAxisDriveInterface".tel2.Input, tel2out := "HydAxisDriveInterface".tel2.Output, tel81in := "HydAxisDriveInterface".tel81.Input, tel81out := "HydAxisDriveInterface".tel81.Output, busy =>, active =>, error =>, status =>, simulatedPosition =>, simulatedForce =>, simulatedVChar =>, forceSensorAnalog_A =>, forceSensorAnalog_B =>)
   END_RUNG
   // the same network as SCL:
   IF "Tag_5" THEN
       "InstHydraulicsSimulationDrive"(enable := true,   // "LSimaHydTO_HydraulicSimulationDrive"
                               minPosition := 0.0,
                               maxPosition := 1000.0,
                               delayTime := 0.02,
                               cycleTime := #CycleTime,
                               vChar_DB_NUMBER := "HydAxisDriveSimulationVChar",
                               axisTO := "SimaHydTO_HydAxis_DRIVE",
                               tel2in := "HydAxisDriveInterface".tel2.Input,
                               tel2out := "HydAxisDriveInterface".tel2.Output,
                               tel81in := "HydAxisDriveInterface".tel81.Input,
                               tel81out := "HydAxisDriveInterface".tel81.Output);
   END_IF;
END_REGION

REGION Network 6
   RUNG wire#powerrail
      "Scale"(Scale_Out => "DENEME".CETVEL)
   END_RUNG
   RUNG wire#powerrail
      Add(in1 := "DENEME".ABSOLUTE_AUX, in2 := "DENEME".OFFSET, out => "DENEME".AbsolutePoz)
   END_RUNG
   // the same network as SCL:
   "Scale"(Scale_Out => "DENEME".CETVEL);
   "DENEME".AbsolutePoz := "DENEME".ABSOLUTE_AUX + "DENEME".OFFSET;
END_REGION

REGION Network 7
   RUNG wire#powerrail
      Contact( "Tag_16" )
      { S7_Templates := "time_type := Time" } "IEC_Timer_0_DB_2".TON(pt := T#10S, et =>)
      Move(in := 10.0, out1 => "DENEME".ABSOLUTE_AUX)
      { S7_Templates := "time_type := Time" } "IEC_Timer_0_DB_1".TON(pt := T#50MS, et =>)
      S_Coil( "step1" )
   END_RUNG
   // the same network as SCL:
   "IEC_Timer_0_DB_2".TON(IN := "Tag_16", PT := T#10S);
   IF "IEC_Timer_0_DB_2".Q THEN "DENEME".ABSOLUTE_AUX := 10.0; END_IF;
   "IEC_Timer_0_DB_1".TON(IN := "IEC_Timer_0_DB_2".Q, PT := T#50MS);
   IF "IEC_Timer_0_DB_1".Q THEN "step1" := TRUE; END_IF;
END_REGION

REGION Network 8
   RUNG wire#powerrail
      Contact( "step1" )
      { S7_Templates := "SrcType := Real" } EQ_Contact(in1 := "DENEME".ABSOLUTE_AUX, in2 := 10.0)
      wire#w1
      R_Coil( "Tag_16" )
   END_RUNG
   RUNG wire#w1
      S_Coil( "step2" )
   END_RUNG
   RUNG wire#w1
      R_Coil( "step1" )
   END_RUNG
   // the same network as SCL:
   IF "step1" AND ("DENEME".ABSOLUTE_AUX = 10.0) THEN
       "Tag_16" := FALSE;
       "step2" := TRUE;
       "step1" := FALSE;
   END_IF;
END_REGION

REGION Network 9
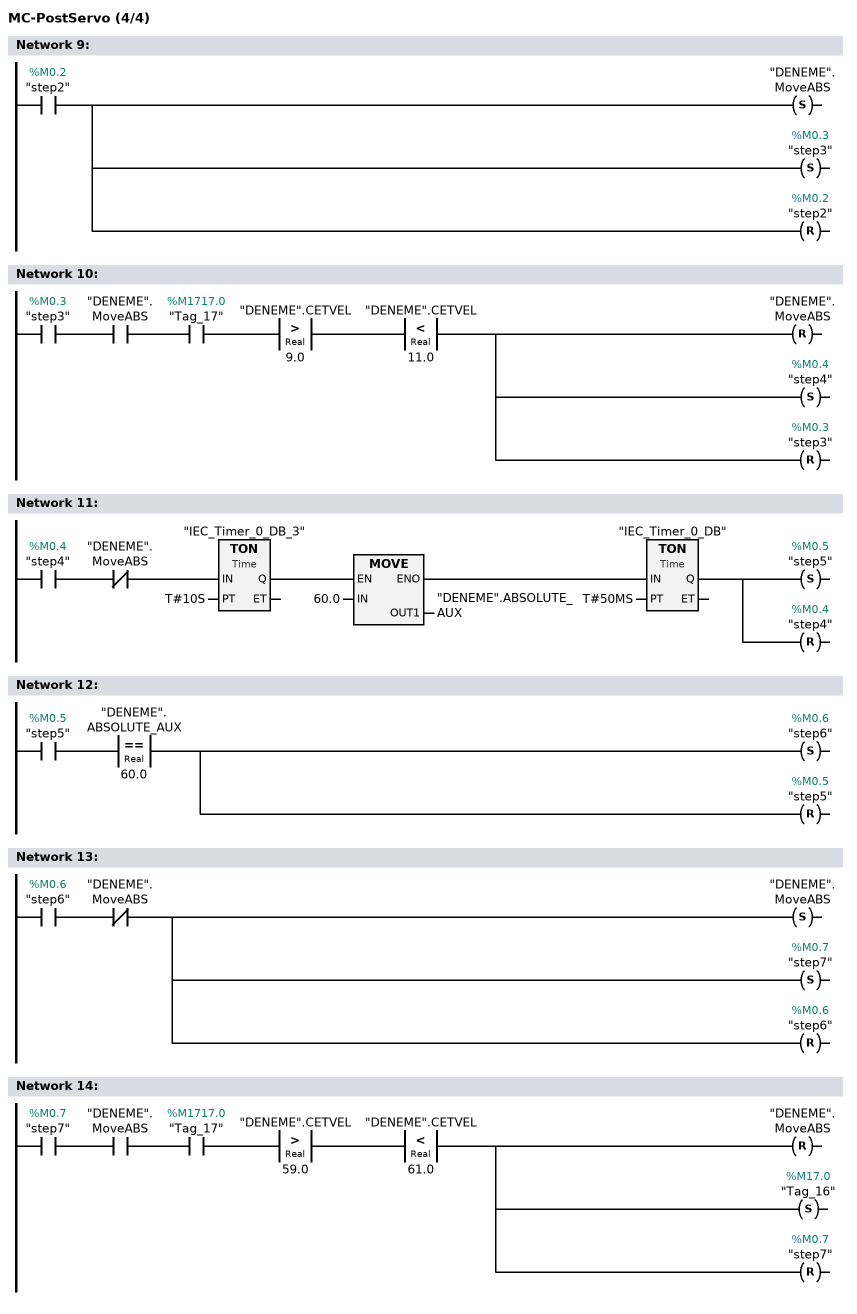
   RUNG wire#powerrail
      Contact( "step2" )
      wire#w1
      S_Coil( "DENEME".MoveABS )
   END_RUNG
   RUNG wire#w1
      S_Coil( "step3" )
   END_RUNG
   RUNG wire#w1
      R_Coil( "step2" )
   END_RUNG
   // the same network as SCL:
   IF "step2" THEN
       "DENEME".MoveABS := TRUE;
       "step3" := TRUE;
       "step2" := FALSE;
   END_IF;
END_REGION

REGION Network 10
   RUNG wire#powerrail
      Contact( "step3" )
      Contact( "DENEME".MoveABS )
      Contact( "Tag_17" )
      { S7_Templates := "SrcType := Real" } GT_Contact(in1 := "DENEME".CETVEL, in2 := 9.0)
      { S7_Templates := "SrcType := Real" } LT_Contact(in1 := "DENEME".CETVEL, in2 := 11.0)
      wire#w1
      R_Coil( "DENEME".MoveABS )
   END_RUNG
   RUNG wire#w1
      S_Coil( "step4" )
   END_RUNG
   RUNG wire#w1
      R_Coil( "step3" )
   END_RUNG
   // the same network as SCL:
   #_w1 := "step3" AND "DENEME".MoveABS AND "Tag_17" AND ("DENEME".CETVEL > 9.0) AND ("DENEME".CETVEL < 11.0);
   IF #_w1 THEN
       "DENEME".MoveABS := FALSE;
       "step4" := TRUE;
       "step3" := FALSE;
   END_IF;
END_REGION

REGION Network 11
   RUNG wire#powerrail
      Contact( "step4" )
      I_Contact( "DENEME".MoveABS )
      { S7_Templates := "time_type := Time" } "IEC_Timer_0_DB_3".TON(pt := T#10S, et =>)
      Move(in := 60.0, out1 => "DENEME".ABSOLUTE_AUX)
      { S7_Templates := "time_type := Time" } "IEC_Timer_0_DB".TON(pt := T#50MS, et =>)
      wire#w1
      S_Coil( "step5" )
   END_RUNG
   RUNG wire#w1
      R_Coil( "step4" )
   END_RUNG
   // the same network as SCL:
   "IEC_Timer_0_DB_3".TON(IN := "step4" AND NOT "DENEME".MoveABS, PT := T#10S);
   IF "IEC_Timer_0_DB_3".Q THEN "DENEME".ABSOLUTE_AUX := 60.0; END_IF;
   "IEC_Timer_0_DB".TON(IN := "IEC_Timer_0_DB_3".Q, PT := T#50MS);
   IF "IEC_Timer_0_DB".Q THEN
       "step5" := TRUE;
       "step4" := FALSE;
   END_IF;
END_REGION

REGION Network 12
   RUNG wire#powerrail
      Contact( "step5" )
      { S7_Templates := "SrcType := Real" } EQ_Contact(in1 := "DENEME".ABSOLUTE_AUX, in2 := 60.0)
      wire#w1
      S_Coil( "step6" )
   END_RUNG
   RUNG wire#w1
      R_Coil( "step5" )
   END_RUNG
   // the same network as SCL:
   IF "step5" AND ("DENEME".ABSOLUTE_AUX = 60.0) THEN
       "step6" := TRUE;
       "step5" := FALSE;
   END_IF;
END_REGION

REGION Network 13
   RUNG wire#powerrail
      Contact( "step6" )
      I_Contact( "DENEME".MoveABS )
      wire#w1
      S_Coil( "DENEME".MoveABS )
   END_RUNG
   RUNG wire#w1
      S_Coil( "step7" )
   END_RUNG
   RUNG wire#w1
      R_Coil( "step6" )
   END_RUNG
   // the same network as SCL:
   #_w1 := "step6" AND NOT "DENEME".MoveABS;
   IF #_w1 THEN
       "DENEME".MoveABS := TRUE;
       "step7" := TRUE;
       "step6" := FALSE;
   END_IF;
END_REGION

REGION Network 14
   RUNG wire#powerrail
      Contact( "step7" )
      Contact( "DENEME".MoveABS )
      Contact( "Tag_17" )
      { S7_Templates := "SrcType := Real" } GT_Contact(in1 := "DENEME".CETVEL, in2 := 59.0)
      { S7_Templates := "SrcType := Real" } LT_Contact(in1 := "DENEME".CETVEL, in2 := 61.0)
      wire#w1
      R_Coil( "DENEME".MoveABS )
   END_RUNG
   RUNG wire#w1
      S_Coil( "Tag_16" )
   END_RUNG
   RUNG wire#w1
      R_Coil( "step7" )
   END_RUNG
   // the same network as SCL:
   #_w1 := "step7" AND "DENEME".MoveABS AND "Tag_17" AND ("DENEME".CETVEL > 59.0) AND ("DENEME".CETVEL < 61.0);
   IF #_w1 THEN
       "DENEME".MoveABS := FALSE;
       "Tag_16" := TRUE;
       "step7" := FALSE;
   END_IF;
END_REGION
END_ORGANIZATION_BLOCK

FUNCTION "LSimaHydTO_MC_SetCharacteristic" : Void
{ S7_Optimized_Access := 'TRUE' }
AUTHOR : APC_ERLF
FAMILY : LSimaHydTO
VERSION : 1.0
   VAR_INPUT 
      valveCharacteristic : DB_ANY;
   END_VAR

   VAR_IN_OUT 
      axis : "LSimaHydTO_typeAxisData";
   END_VAR

   VAR CONSTANT 
      NO_ALARM : Word := 0;
   END_VAR


BEGIN
	//================================================================================
	//SIEMENS AG // (c)Copyright 2019 All Rights Reserved
	//--------------------------------------------------------------------------------
	//Library:       LSimaHydTO
	//Tested with:   S7-15xx
	//Engineering:   TIA Portal  V15
	//Restrictions:  -
	//Requirements:  S7-1500 (FW 2.5)
	//Functionality: Set characteristics for axis
	//
	//--------------------------------------------------------------------------------
	//Change log table:
	//
	//Version     Date          Expert in charge    Changes applied
	//01.00.00    15.03.2018    APC_ERLF            First released version
	//================================================================================
	
	#axis.ValveCharacteristic.DB_NUMBER := DB_ANY_TO_UINT(#valveCharacteristic);
	
END_FUNCTION

FUNCTION_BLOCK "LSimaHydTO_HydAxisCall"
{ S7_Optimized_Access := 'TRUE' }
AUTHOR : APC_ERLF
FAMILY : LSimaHydTO
VERSION : 1.0
   VAR_INPUT 
      axisTO { ExternalAccessible := 'False'; ExternalVisible := 'False'; ExternalWritable := 'False'} : DB_ANY;
      pressure_A_RawValue { ExternalAccessible := 'False'; ExternalVisible := 'False'; ExternalWritable := 'False'} : Word;
      pressure_B_RawValue { ExternalAccessible := 'False'; ExternalVisible := 'False'; ExternalWritable := 'False'} : Word;
      cycleTime { ExternalAccessible := 'False'; ExternalVisible := 'False'; ExternalWritable := 'False'} : UDInt;
   END_VAR

   VAR_OUTPUT 
      error { ExternalAccessible := 'False'; ExternalVisible := 'False'; ExternalWritable := 'False'} : Bool;
   END_VAR

   VAR_IN_OUT 
      axisData : "LSimaHydTO_typeAxisData";
   END_VAR

   VAR 
      statInit { ExternalAccessible := 'False'; ExternalVisible := 'False'; ExternalWritable := 'False'} : Bool := true;
      statTypeOfAxis { ExternalAccessible := 'False'; ExternalVisible := 'False'; ExternalWritable := 'False'} : Int;
      instHydAxisFB { ExternalAccessible := 'False'; ExternalVisible := 'False'; ExternalWritable := 'False'} : "LSimaHydTO_HydAxis";
      instHydSyncAxisFB { ExternalAccessible := 'False'; ExternalVisible := 'False'; ExternalWritable := 'False'} : "LSimaHydTO_HydSyncAxis";
   END_VAR

   VAR CONSTANT 
      SPEED_AXIS : Int;
      POS_AXIS : Int := 1;
      SYNC_AXIS : Int := 2;
      ERROR_REACTION_DISABLE : DInt := 4;
      ALARM_TO_TYPE : UDInt := 9101;
   END_VAR


BEGIN
	//=============================================================================
	//SIEMENS AG
	//(c)Copyright 2016 All Rights Reserved
	//-----------------------------------------------------------------------------
	//Library:       SimaHydTO_HMI
	//Tested with:   S7-1500 V2.5
	//Engineering:   TIA Portal V15
	// Restrictions:  Call in PosServo OB
	// Requirements:  S7-1500 (FW 2.5) TO positioning or synchronous axis
	// Functionality: Function block call of FB "HydAxis"
	//-----------------------------------------------------------------------------
	// Change log table:
	// Version  Date       Expert in charge Changes applied
	//01.00.00    05.03.2019    APC_ERLF            First released version
	//=============================================================================
	
	
	IF #statInit THEN
	  #error := FALSE;
	  #axisData.TO_Axis := #axisTO;
	  //TO PositioningAxis
	  IF TypeOfDB(#axisTO) = TO_PositioningAxis THEN
	    #statTypeOfAxis := #POS_AXIS;
	    //TO SynchronousAxis
	  ELSIF TypeOfDB(#axisTO) = TO_SynchronousAxis THEN
	    #statTypeOfAxis := #SYNC_AXIS;
	    //TO SpeedAxis
	  ELSE
	    #statTypeOfAxis := #SPEED_AXIS;
	  END_IF;
	  #instHydAxisFB.cycleTime := #cycleTime;
	  #statInit := FALSE;
	END_IF;
	
	#instHydAxisFB.pressure_A_RawValue := #pressure_A_RawValue;
	#instHydAxisFB.pressure_B_RawValue := #pressure_B_RawValue;
	
	CASE #statTypeOfAxis OF
	    
	  #POS_AXIS:
	    #instHydAxisFB(axisTO := #axisTO,
	                   axisData := #axisData);
	    
	  #SYNC_AXIS:
	    #instHydSyncAxisFB(axisTO := #axisTO,
	                       axisData := #axisData,
	                       instHydAxisFB := #instHydAxisFB);
	  ELSE
	    //Error - Wrong axis type
	    #axisData.ErrorWord.%X1 := TRUE;
	    #axisData.ErrorDetail.Number := #ALARM_TO_TYPE;
	    #axisData.ErrorDetail.Reaction := #ERROR_REACTION_DISABLE;
	    #error := TRUE;
	END_CASE;
	
END_FUNCTION_BLOCK

FUNCTION_BLOCK "LSimaHydTO_HydAxis"
{ S7_Optimized_Access := 'TRUE' }
AUTHOR : APC_ERLF
FAMILY : LSimaHydTO
VERSION : 1.22
   VAR_INPUT 
      pressure_A_RawValue { ExternalAccessible := 'False'; ExternalVisible := 'False'; ExternalWritable := 'False'} : Word;
      pressure_B_RawValue { ExternalAccessible := 'False'; ExternalVisible := 'False'; ExternalWritable := 'False'} : Word;
      cycleTime { ExternalAccessible := 'False'; ExternalVisible := 'False'; ExternalWritable := 'False'} : UDInt;
   END_VAR

   VAR_IN_OUT 
      axisTO {InstructionName := 'TO_PositioningAxis'; LibVersion := '4.0'} : TO_PositioningAxis;
      axisData : "LSimaHydTO_typeAxisData";
   END_VAR

   VAR 
      statSampleTime { ExternalAccessible := 'False'; ExternalVisible := 'False'; ExternalWritable := 'False'} : LReal;
      statInit { ExternalAccessible := 'False'; ExternalVisible := 'False'; ExternalWritable := 'False'} : Bool := TRUE;
      statAxisState { ExternalAccessible := 'False'; ExternalVisible := 'False'; ExternalWritable := 'False'} : DInt;
      statAxisStateNext { ExternalAccessible := 'False'; ExternalVisible := 'False'; ExternalWritable := 'False'} : DInt;
      statAxisStateOld { ExternalAccessible := 'False'; ExternalVisible := 'False'; ExternalWritable := 'False'} : DInt;
      statPosCtrlOld { ExternalAccessible := 'False'; ExternalVisible := 'False'; ExternalWritable := 'False'} : Bool;
      statForceCtrlOld { ExternalAccessible := 'False'; ExternalVisible := 'False'; ExternalWritable := 'False'} : Bool;
      statForceLimOld { ExternalAccessible := 'False'; ExternalVisible := 'False'; ExternalWritable := 'False'} : Bool;
      statForceLimitingVelNorm { ExternalAccessible := 'False'; ExternalVisible := 'False'; ExternalWritable := 'False'} : LReal;
      statForceLimIntPos { ExternalAccessible := 'False'; ExternalVisible := 'False'; ExternalWritable := 'False'} : LReal;
      statVCharOld { ExternalAccessible := 'False'; ExternalVisible := 'False'; ExternalWritable := 'False'} : UInt := 0;
      statQOutput { ExternalAccessible := 'False'; ExternalVisible := 'False'; ExternalWritable := 'False'} : LReal;
      statQOutputOld { ExternalAccessible := 'False'; ExternalVisible := 'False'; ExternalWritable := 'False'} : LReal;
      statCtrlOutUppLimit { ExternalAccessible := 'False'; ExternalVisible := 'False'; ExternalWritable := 'False'} : LReal := 1000000000000.0;
      statCtrlOutLowLimit { ExternalAccessible := 'False'; ExternalVisible := 'False'; ExternalWritable := 'False'} : LReal := -1000000000000.0;
      statActualNorm { ExternalAccessible := 'False'; ExternalVisible := 'False'; ExternalWritable := 'False'} : "LSimaHydTO_typeMotionVector";
      statCommandNorm { ExternalAccessible := 'False'; ExternalVisible := 'False'; ExternalWritable := 'False'} : "LSimaHydTO_typeMotionVector";
      instVelSmoothingFilter { ExternalAccessible := 'False'; ExternalVisible := 'False'; ExternalWritable := 'False'} : "LSimaHydTO_T1";
      instAccSmoothingFilter { ExternalAccessible := 'False'; ExternalVisible := 'False'; ExternalWritable := 'False'} : "LSimaHydTO_T1";
      instVCharSmoothing { ExternalAccessible := 'False'; ExternalVisible := 'False'; ExternalWritable := 'False'} : "LSimaHydTO_T1";
      instBalancePos { ExternalAccessible := 'False'; ExternalVisible := 'False'; ExternalWritable := 'False'} : "LSimaHydTO_T1";
      instBalanceForce { ExternalAccessible := 'False'; ExternalVisible := 'False'; ExternalWritable := 'False'} : "LSimaHydTO_T1";
      instPositionController { ExternalAccessible := 'False'; ExternalVisible := 'False'; ExternalWritable := 'False'} : "LSimaHydTO_PIDT1";
      instForceController { ExternalAccessible := 'False'; ExternalVisible := 'False'; ExternalWritable := 'False'} : "LSimaHydTO_PIDT1";
      statForceLimitation { ExternalAccessible := 'False'; ExternalVisible := 'False'; ExternalWritable := 'False'} : Bool;
      statInternalStop { ExternalAccessible := 'False'; ExternalVisible := 'False'; ExternalWritable := 'False'} : Bool;
      statNumOfLoop { ExternalAccessible := 'False'; ExternalVisible := 'False'; ExternalWritable := 'False'} : Int;
      statCmdPosOld { ExternalAccessible := 'False'; ExternalVisible := 'False'; ExternalWritable := 'False'} : LReal;
      statForceProfileTime { ExternalAccessible := 'False'; ExternalVisible := 'False'; ExternalWritable := 'False'} : LReal;
      statForceConditionActive { ExternalAccessible := 'False'; ExternalVisible := 'False'; ExternalWritable := 'False'} : Bool;
      statConditionMode { ExternalAccessible := 'False'; ExternalVisible := 'False'; ExternalWritable := 'False'} : DInt;
      statCompareMode { ExternalAccessible := 'False'; ExternalVisible := 'False'; ExternalWritable := 'False'} : DInt;
      statConditionValue { ExternalAccessible := 'False'; ExternalVisible := 'False'; ExternalWritable := 'False'} : LReal;
      statVelocityLimitingValueNorm { ExternalAccessible := 'False'; ExternalVisible := 'False'; ExternalWritable := 'False'} : LReal;
      statInProfileOld { ExternalAccessible := 'False'; ExternalVisible := 'False'; ExternalWritable := 'False'} : Bool;
      statForceCtrlCondition { ExternalAccessible := 'False'; ExternalVisible := 'False'; ExternalWritable := 'False'} : Bool;
      statManEnableOld { ExternalAccessible := 'False'; ExternalVisible := 'False'; ExternalWritable := 'False'} : Bool;
      statForceCtrCmdValueOld { ExternalAccessible := 'False'; ExternalVisible := 'False'; ExternalWritable := 'False'} : LReal;
      statForceProfileDB { ExternalAccessible := 'False'; ExternalVisible := 'False'; ExternalWritable := 'False'} : DB_ANY;
      statVCharDB { ExternalAccessible := 'False'; ExternalVisible := 'False'; ExternalWritable := 'False'} : DB_ANY;
      statErrorVariant { ExternalAccessible := 'False'; ExternalVisible := 'False'; ExternalWritable := 'False'} : Int;
      statMotionSetPointNorm { ExternalAccessible := 'False'; ExternalVisible := 'False'; ExternalWritable := 'False'} : LReal;
      statForceCtrlActive { ExternalAccessible := 'False'; ExternalVisible := 'False'; ExternalWritable := 'False'} : Bool;
      statManQOutput { ExternalAccessible := 'False'; ExternalVisible := 'False'; ExternalWritable := 'False'} : LReal;
      statReqForward { ExternalAccessible := 'False'; ExternalVisible := 'False'; ExternalWritable := 'False'} : Bool;
      statReqBackward { ExternalAccessible := 'False'; ExternalVisible := 'False'; ExternalWritable := 'False'} : Bool;
      instValvesControl { ExternalAccessible := 'False'; ExternalVisible := 'False'; ExternalWritable := 'False'} : "LSimaHydTO_ValvesControl";
      statRampingForward { ExternalAccessible := 'False'; ExternalVisible := 'False'; ExternalWritable := 'False'} : Bool;
      statRampingBackward { ExternalAccessible := 'False'; ExternalVisible := 'False'; ExternalWritable := 'False'} : Bool;
      statManOutDeceleration { ExternalAccessible := 'False'; ExternalVisible := 'False'; ExternalWritable := 'False'} : Bool;
      statDecelerationDistance { ExternalAccessible := 'False'; ExternalVisible := 'False'; ExternalWritable := 'False'} : LReal;
      statManRamp { ExternalAccessible := 'False'; ExternalVisible := 'False'; ExternalWritable := 'False'} : LReal;
      statElapsedDelayTime { ExternalAccessible := 'False'; ExternalVisible := 'False'; ExternalWritable := 'False'} : LReal;
      statForceCtrlSetPointNorm { ExternalAccessible := 'False'; ExternalVisible := 'False'; ExternalWritable := 'False'} : LReal;
      statStatusWordMaskedOld { ExternalAccessible := 'False'; ExternalVisible := 'False'; ExternalWritable := 'False'} : DWord;
      instMC_MOVEVELOCITY_Zero {InstructionName := 'MC_MOVEVELOCITY'; LibVersion := '4.0'; ExternalAccessible := 'False'; ExternalVisible := 'False'; ExternalWritable := 'False'} : MC_MOVEVELOCITY;
      instMC_VELOCITY_Zero_ForceCtrl {InstructionName := 'MC_MOVEVELOCITY'; LibVersion := '4.0'; ExternalAccessible := 'False'; ExternalVisible := 'False'; ExternalWritable := 'False'} : MC_MOVEVELOCITY;
      statForceDirPos { ExternalAccessible := 'False'; ExternalVisible := 'False'; ExternalWritable := 'False'} : Bool;
      statAxisTOStatusWord { ExternalAccessible := 'False'; ExternalVisible := 'False'; ExternalWritable := 'False'} : DWord;
      statAxisTOErrorWord { ExternalAccessible := 'False'; ExternalVisible := 'False'; ExternalWritable := 'False'} : DWord;
      statDynamicLimits { ExternalAccessible := 'False'; ExternalVisible := 'False'; ExternalWritable := 'False'} : "LSimaHydTO_typeDynamicLimits";
      statExecuteMovement { ExternalAccessible := 'False'; ExternalVisible := 'False'; ExternalWritable := 'False'} : Bool;
      statEnable { ExternalAccessible := 'False'; ExternalVisible := 'False'; ExternalWritable := 'False'} : Bool;
      instMC_HALT {InstructionName := 'MC_HALT'; LibVersion := '4.0'; ExternalAccessible := 'False'; ExternalVisible := 'False'; ExternalWritable := 'False'} : MC_HALT;
      statIntForceFactor { ExternalAccessible := 'False'; ExternalVisible := 'False'; ExternalWritable := 'False'} : LReal := 0.1;
      statIntVelocityFactor { ExternalAccessible := 'False'; ExternalVisible := 'False'; ExternalWritable := 'False'} : LReal := 1.0;
      statExtError { ExternalAccessible := 'False'; ExternalVisible := 'False'; ExternalWritable := 'False'} : Bool;
      statAutoReset { ExternalAccessible := 'False'; ExternalVisible := 'False'; ExternalWritable := 'False'} : Bool;
      statManPosCtrlOld { ExternalAccessible := 'False'; ExternalVisible := 'False'; ExternalWritable := 'False'} : Bool;
      statQOutputMan { ExternalAccessible := 'False'; ExternalVisible := 'False'; ExternalWritable := 'False'} : LReal;
      statQOutMax { ExternalAccessible := 'False'; ExternalVisible := 'False'; ExternalWritable := 'False'} : LReal := 100.0;
      statForceCommand { ExternalAccessible := 'False'; ExternalVisible := 'False'; ExternalWritable := 'False'} : "LSimaHydTO_typeInternalControlForceCmd";
      statConditionTime { ExternalAccessible := 'False'; ExternalVisible := 'False'; ExternalWritable := 'False'} : LReal;
      statForceLimPosCmd { ExternalAccessible := 'False'; ExternalVisible := 'False'; ExternalWritable := 'False'} : LReal;
      statInLimitationOld { ExternalAccessible := 'False'; ExternalVisible := 'False'; ExternalWritable := 'False'} : Bool;
      statFolErMin { ExternalAccessible := 'False'; ExternalVisible := 'False'; ExternalWritable := 'False'} : LReal;
      statFolErMax { ExternalAccessible := 'False'; ExternalVisible := 'False'; ExternalWritable := 'False'} : LReal;
      statPosWindow { ExternalAccessible := 'False'; ExternalVisible := 'False'; ExternalWritable := 'False'} : LReal;
      instWriteAxisSetpoint { ExternalAccessible := 'False'; ExternalVisible := 'False'; ExternalWritable := 'False'} : "LSimaHydTO_WriteAxisSetpoint";
      statClamping { ExternalAccessible := 'False'; ExternalVisible := 'False'; ExternalWritable := 'False'} : Bool;
      statRetVCHar { ExternalAccessible := 'False'; ExternalVisible := 'False'; ExternalWritable := 'False'} : LReal;
      statAdaption { ExternalAccessible := 'False'; ExternalVisible := 'False'; ExternalWritable := 'False'} : Bool := TRUE;
      instAxisAlarm {InstructionName := 'Program_Alarm'; LibVersion := '1.0'; ExternalAccessible := 'False'; ExternalVisible := 'False'; ExternalWritable := 'False'} : Program_Alarm;
      statErrInternal { ExternalAccessible := 'False'; ExternalVisible := 'False'; ExternalWritable := 'False'} : Bool;
      statErrInternalOld { ExternalAccessible := 'False'; ExternalVisible := 'False'; ExternalWritable := 'False'} : Bool;
      statErrAddValue { ExternalAccessible := 'False'; ExternalVisible := 'False'; ExternalWritable := 'False'} : Int;
      statInstName { ExternalAccessible := 'False'; ExternalVisible := 'False'; ExternalWritable := 'False'} : WString[80];
      statAxisTOErrorReaction { ExternalAccessible := 'False'; ExternalVisible := 'False'; ExternalWritable := 'False'} : DInt;
      statSmoothRamp { ExternalAccessible := 'False'; ExternalVisible := 'False'; ExternalWritable := 'False'} : LReal;
      statSmoothRampOut { ExternalAccessible := 'False'; ExternalVisible := 'False'; ExternalWritable := 'False'} : LReal;
      statSmoothingModeOld { ExternalAccessible := 'False'; ExternalVisible := 'False'; ExternalWritable := 'False'} : Int;
      statForceUnit { ExternalAccessible := 'False'; ExternalVisible := 'False'; ExternalWritable := 'False'} : UDInt;
      statLengthUnit { ExternalAccessible := 'False'; ExternalVisible := 'False'; ExternalWritable := 'False'} : UDInt;
      statVelocityUnit { ExternalAccessible := 'False'; ExternalVisible := 'False'; ExternalWritable := 'False'} : UDInt;
      statHomingDoneOld { ExternalAccessible := 'False'; ExternalVisible := 'False'; ExternalWritable := 'False'} : Bool;
      statMaxSetPoint { ExternalAccessible := 'False'; ExternalVisible := 'False'; ExternalWritable := 'False'} : LReal;
   END_VAR

   VAR_TEMP 
      tempRampGenActive : Bool;
      tempCompareValue : LReal;
      tempInProfile : Bool;
      tempVCharVar : Variant;
      tempForceProfileVar : Variant;
      tempQOutput : LReal;
      tempManualSafetyDistance : LReal;
      tempRefToVChar : REF_TO "LSimaHydTO_typeVCharData";
      tempRefToForceProfile : REF_TO "LSimaHydTO_typeProfile";
      tempStatusWordMasked : DWord;
      tempChangePosCtrl : Bool;
      tempAbortMovement : Bool;
      tempSmoothingMode : Int;
      tempActualVelocity : LReal;
      tempAccFactor : LReal;
   END_VAR

